// TwinCAT 3 PLC project Library
// Title: lcls-twincat-motion
// Company: SLAC
// ProjectVersion: 0.0.0
// ProgramVersion: 3.1.4026.15
// libraries:
//   LCLS General, * (SLAC)
//   lcls-twincat-math, * (SLAC - LCLS)
//   PMPS, * (SLAC - LCLS)
//   Tc2_EtherCAT, * (Beckhoff Automation GmbH)
//   Tc2_Math, * (Beckhoff Automation GmbH)
//   Tc2_MC2, * (Beckhoff Automation GmbH)
//   Tc2_Standard, * (Beckhoff Automation GmbH)
//   Tc2_System, * (Beckhoff Automation GmbH)
//   Tc2_Utilities, * (Beckhoff Automation GmbH)
//   Tc3_IPCDiag, * (Beckhoff Automation GmbH)
//   Tc3_JsonXml, * (Beckhoff Automation GmbH)
//   Tc3_Module, * (Beckhoff Automation GmbH)
//   TcUnit, * (www.tcunit.org)
// project tree:
//   DUTs/Deprecated/ ENUM_MotionRequest.TcDUT (not stored), DUT_MotionPneumaticActuator.TcDUT (not stored), DUT_MotionStage.TcDUT (not stored), DUT_PositionState.TcDUT (not stored), EL5042_Status.TcDUT (not stored), ENUM_EpicsHomeCmd.TcDUT (not stored), ENUM_EpicsInOut.TcDUT (not stored), ENUM_EpicsInOut_INT.TcDUT (not stored), ENUM_EpicsMotorCmd.TcDUT (not stored), ENUM_MotionFFType.TcDUT (not stored), ENUM_PnuematicActuatorPositionState.TcDUT (not stored), ENUM_StageBrakeMode.TcDUT (not stored), ENUM_StageEnableMode.TcDUT (not stored), ENUM_StatePMPSStatus.TcDUT (not stored)
//   DUTs/ ST_AxisParameterSetExposed.TcDUT (not stored), E_LCLSMotionError.TcDUT (not stored), E_MotionFFType.TcDUT (not stored), E_StatePMPSStatus.TcDUT (not stored), ST_MotionDrive.TcDUT (not stored), ST_MotionStage.TcDUT (not stored), ST_MotionEpicsInterface.TcDUT (not stored), ST_PositionState.TcDUT, ST_StateEpicsToPlc.TcDUT (not stored), ST_StatePlcToEpics.TcDUT (not stored), ST_StatePMPSEpicsToPlc.TcDUT (not stored), ST_EL5042_Status.TcDUT (not stored), E_EpicsHomeCmd.TcDUT (not stored), E_EpicsInOut.TcDUT (not stored), E_EpicsMotorCmd.TcDUT (not stored), E_MotionRequest.TcDUT (not stored), E_StageBrakeMode.TcDUT (not stored), E_StageEnableMode.TcDUT (not stored), ST_MotionPneumaticActuator.TcDUT (not stored), E_PnuematicActuatorPositionState.TcDUT (not stored), ST_RenishawAbsEnc.TcDUT (not stored), ST_StatePMPSPlcToEpics.TcDUT (not stored)
//   GVLs/ MOTION_GVL.TcGVL (not stored), MotionConstants.TcGVL (not stored)
//   / PlcTask.TcTTO (not stored)
//   POUs/Deprecated/ FB_EpicsInOut.TcPOU (not stored), FB_PositionStateBase.TcPOU (not stored), FB_PositionStateBase_WithPMPS.TcPOU (not stored), FB_PositionStateBase_WithPMPS_Test.TcPOU (not stored), FB_PositionStateInOut.TcPOU (not stored), FB_PositionStateInOut_WithPMPS.TcPOU (not stored), FB_PositionStateInOut_WithPMPS_Test.TcPOU (not stored), FB_PositionStateManager.TcPOU (not stored), FB_PositionStatePMPS.TcPOU (not stored), FB_PositionStatePMPS_Base.TcPOU (not stored), FB_PositionStatePMPS_Test.TcPOU (not stored), FB_StatePTPMove.TcPOU (not stored)
//   POUs/ImplicitChecks/ CheckBounds.TcPOU (not stored), CheckDivDInt.TcPOU (not stored), CheckDivLInt.TcPOU (not stored), CheckDivLReal.TcPOU (not stored), CheckDivReal.TcPOU (not stored)
//   POUs/Motion/ FB_EncoderValue.TcPOU (not stored), FB_EncSaveRestore.TcPOU (not stored), FB_LogMotionError.TcPOU (not stored), FB_MotionAxisDS402.TcPOU, FB_MotionAxisDS402NC.TcPOU, FB_MotionAxisNC.TcPOU, FB_MotionAxisNCContinuous.TcPOU, FB_MotionBacklashCompensation.TcPOU (not stored), FB_MotionDrive.TcPOU (not stored), FB_MotionHoming.TcPOU (not stored), FB_MotionRequest.TcPOU (not stored), FB_MotionStage.TcPOU (not stored), FB_MotionStageNCParams.TcPOU (not stored), FB_MotionStageSim.TcPOU (not stored), FB_MotionPneumaticActuator.TcPOU (not stored), FB_MotionVirtualFrame.TcPOU (not stored), FB_MotionAxisPneumatic.TcPOU
//   POUs/Motion/Gantry/ FB_GantryAutoCoupling.TcPOU (not stored), FB_GantryDiffVirtualLimitSwitch.TcPOU (not stored)
//   POUs/Motion/ITFs/ I_Brake.TcIO (not stored), I_MotionAxisContinuous.TcIO, I_MotionInterlocks.TcIO (not stored), I_MotionLogger.TcIO (not stored), I_MotionDrive.TcIO, I_MotionAxis.TcIO, I_PersistantDataStorage.TcIO (not stored)
//   POUs/Motion/PMPS/ FB_EncErrorFFO.TcPOU (not stored), FB_MiscStatesErrorFFO.TcPOU (not stored), FB_MotionBPTM.TcPOU (not stored), FB_MotionClearAsserts.TcPOU (not stored), FB_MotionReadPMPSDBND.TcPOU (not stored), FB_PerMotorFFOND.TcPOU (not stored), FB_NCErrorFFO.TcPOU (not stored), FB_PositionStatePMPS1D.TcPOU (not stored), FB_PositionStatePMPS2D.TcPOU (not stored), FB_PositionStatePMPS3D.TcPOU (not stored), FB_PositionStatePMPSND_Core.TcPOU (not stored), FB_Standard_PMPSDB.TcPOU (not stored), FB_StatePMPSEnables.TcPOU (not stored), FB_StatePMPSEnablesND.TcPOU (not stored)
//   POUs/Motion/States/Examples/ FB_PositionState1D_InOut.TcPOU (not stored), FB_PositionStatePMPS2D_InOut.TcPOU (not stored), FB_PositionStatePMPS1D_InOut.TcPOU (not stored), FB_PositionState2D_InOut.TcPOU (not stored)
//   POUs/Motion/States/ FB_PositionState2D.TcPOU (not stored), FB_PositionState3D.TcPOU (not stored), FB_PositionStateND_Core.TcPOU (not stored), FB_PositionStateMove.TcPOU (not stored), FB_PositionState1D.TcPOU (not stored), FB_PositionStateMoveND.TcPOU, FB_PositionStateRead.TcPOU (not stored), FB_PositionStateReadND.TcPOU (not stored), FB_StateSetupHelper.TcPOU (not stored), FB_StatesInputHandler.TcPOU (not stored)
//   POUs/Motion/States/Helpers/ FB_RawCountConverter.TcPOU (not stored), F_AtPositionState.TcPOU (not stored), F_PosOverLowerBound.TcPOU (not stored), F_PosUnderUpperBound.TcPOU (not stored), F_PosWithinDelta.TcPOU (not stored)
//   POUs/Motion/States/Internals/ FB_PositionStateInternal.TcPOU (not stored), FB_PositionStateInternalND.TcPOU (not stored), FB_PositionStateLock.TcPOU (not stored)
//   POUs/Motion/Utils/ FB_SetEnables.TcPOU (not stored), F_MotionErrorCodeLookup.TcPOU (not stored)
//   POUs/MotorTesting/ FB_MicroStepCountTest.TcPOU (not stored)
//   tc_mca_std_lib/DUTs/ DUT_AxisStatus_v0_01.TcDUT (not stored)
//   tc_mca_std_lib/GVLs/ GVL.TcGVL (not stored)
//   tc_mca_std_lib/POUs/ChangeConfig/ FB_ReadFloatParameter.TcPOU (not stored), FB_ReadParameterInNc_v1_00.TcPOU (not stored), FB_WriteFloatParameter.TcPOU (not stored), FB_WriteParameterInNc_v1_00.TcPOU (not stored)
//   tc_mca_std_lib/POUs/ErrorHandling/ DUT_ErrorState.TcDUT (not stored), DUT_TerminalError.TcDUT (not stored), FB_ErrorList.TcPOU (not stored), FB_TerminalError.TcPOU (not stored), GVL_ErrorSystem.TcGVL (not stored), ST_ErrorSystem.TcDUT (not stored)
//   tc_mca_std_lib/POUs/Hardware/EtherCAT_Terminals/Analog_Inputs/ EL3174_0002.TcPOU (not stored), EL3214.TcPOU (not stored), EL3255.TcPOU (not stored), FB_CalculateFrequency_3702_v0_01.TcPOU (not stored)
//   tc_mca_std_lib/POUs/Hardware/EtherCAT_Terminals/Digital_Inputs/ EL1008.TcPOU (not stored), EL1018.TcPOU (not stored), EL1808.TcPOU (not stored), EL1809.TcPOU (not stored), EL1819.TcPOU (not stored), FB_EL1252ASM_v1_00.TcPOU (not stored)
//   tc_mca_std_lib/POUs/Hardware/EtherCAT_Terminals/Digital_Outputs/ EL2014.TcPOU (not stored), EL2252.TcPOU (not stored), EL2808.TcPOU (not stored), EL2819.TcPOU (not stored)
//   tc_mca_std_lib/POUs/Hardware/EtherCAT_Terminals/Digital_Outputs/External_Types/ dutEL2521_Ctrl.TcDUT (not stored), dutEL2521_Status.TcDUT (not stored)
//   tc_mca_std_lib/POUs/Hardware/EtherCAT_Terminals/Measuring_Terminals/ EL5002.TcPOU (not stored), EL5021.TcPOU (not stored), EL5042.TcPOU (not stored), EL5101.TcPOU (not stored)
//   tc_mca_std_lib/POUs/Hardware/EtherCAT_Terminals/Motion/ EL7211_v1_00.TcPOU (not stored), EL9576_v1_00.TcPOU (not stored)
//   tc_mca_std_lib/POUs/Hardware/EtherCAT_Terminals/System/ EL9410.TcPOU (not stored), EL9505.TcPOU (not stored)
//   tc_mca_std_lib/POUs/Hardware/Other/ EK1200.TcPOU (not stored)
//   tc_mca_std_lib/POUs/Motion/ FB_DriveVirtual.TcPOU (not stored), FB_NcAxis.TcPOU (not stored)
//   tc_mca_std_lib/POUs/Motion/Homing/ FB_HomeDirect.TcPOU (not stored), FB_HomeFinish.TcPOU (not stored), FB_HomePrepare.TcPOU (not stored), FB_HomeReadNcVelocities.TcPOU (not stored), FB_HomeReadSoftLimEnable.TcPOU (not stored), FB_HomeToSwitch.TcPOU (not stored), FB_HomeVirtual.TcPOU (not stored), FB_HomeWriteNcVelocities.TcPOU (not stored), FB_HomeWriteSoftLimEnable.TcPOU (not stored)
//   Tests/ FB_AtPositionState_Test.TcPOU (not stored), FB_AxisParameterSetExposed_Test.TcPOU (not stored), FB_MiscStatesErrorFFO_Test.TcPOU (not stored), FB_MotionAxisNC_Test.TcPOU, FB_MotionAxisNCContinuous_Test.TcPOU, FB_MotionBPTM_Test.TcPOU (not stored), FB_MotionClearAsserts_Test.TcPOU (not stored), FB_MotionReadPMPSDBND_Test.TcPOU (not stored), FB_MotionVirtualFrame_Test.TcPOU (not stored), FB_NCErrorFFO_Test.TcPOU (not stored), FB_PerMotorFFOND_Test.TcPOU (not stored), FB_PositionStateMoveND_Test.TcPOU (not stored), FB_PositionStateMove_Test.TcPOU (not stored), FB_PositionStatePMPSND_Test.TcPOU (not stored), FB_PositionStateReadND_Test.TcPOU (not stored), FB_PositionStateRead_Test.TcPOU (not stored), FB_PositionStateND_Test.TcPOU (not stored), FB_PowerEnableMode_Test.TcPOU (not stored), FB_MotionBacklashCompensation_Test.TcPOU (not stored), FB_StatePMPSEnablesND_Test.TcPOU (not stored), FB_StatePMPSEnables_Test.TcPOU (not stored), FB_StateSetupHelper_Test.TcPOU (not stored), FB_TestHelperSetAndMove_Test.TcPOU (not stored), FB_TestStateInitTiming.TcPOU (not stored), PRG_TEST.TcPOU
//   Tests/Helpers/ E_TestStates.TcDUT (not stored), FB_CauseNCError.TcPOU (not stored), FB_MotionStageSetAndMoveHelper.TcPOU (not stored), FB_MotionStageSetHelper.TcPOU (not stored), FB_MotorTestSuite.TcPOU (not stored), FB_PMPSJsonTestHelper.TcPOU (not stored), FB_TestHelperSetAndMove.TcPOU (not stored)
//   Tests/TestDoubles/ FB_MotionAxisNCTestDouble.TcPOU
//   Version/ Global_Version.TcGVL (not stored)

// ---- DUTs/ST_PositionState.TcDUT
TYPE ST_PositionState :
    // Defines settings and current safety status for moves to specific positions for an axis
STRUCT
    // Name as queried via the NAME PV in EPICS
    {attribute 'pytmc' := '
        pv: NAME
        io: input
        field: DESC Name of this position state
    '}
    sName: STRING := 'Invalid';

    // Position associated with this state
    {attribute 'pytmc' := '
        pv: SETPOINT
        io: io
        field: DESC Axis position associated with this state
    '}
    fPosition: LREAL;

    {attribute 'pytmc' := '
        pv: ENCODER
        io: i
        field: DESC Encoder count associated with this state
    '}
    nEncoderCount: UDINT;

    // Maximum allowable deviation from fPosition while at the state
    fDelta: LREAL;

    // Speed at which to move to this state
    {attribute 'pytmc' := '
        pv: VELO
        io: io
        field: DESC Speed at which to move to this state
    '}
    fVelocity: LREAL;

    // (optional) Acceleration to use for moves to this state
    fAccel: LREAL;

    // (optional) Deceleration to use for moves to this state
    fDecel: LREAL;

    // Safety parameter. This must be set to TRUE by the PLC program to allow moves to this state. This is expected to change as conditions change.
    {attribute 'pytmc' := '
        pv: MOVE_OK
        io: i
        field: ZNAM FALSE
        field: ONAM TRUE
        field: DESC TRUE if the move would be safe
    '}
    bMoveOk: BOOL;

    // Signifies to FB_PositionStateLock that this state should be immutable
    bLocked: BOOL;

    // Set this to TRUE when you make your state. This defaults to FALSE so that uninitialized states can never be moved to
    bValid: BOOL;

    // Set this to TRUE when you want to use the raw encoder counts to define the state
    bUseRawCounts: BOOL;

    // Is set to TRUE by FB_PositionStateInternal when called
    bUpdated: BOOL;

    // We give this a state name and it is used to load parameters from the pmps database.
    stPMPS: ST_DbStateParams;

    // Set true on the rising trigger for execution of a state mover.
    // Used to sequence movement of a individual axes in a multiple state mover.
    {attribute 'pytmc' := '
        pv: PLC:bMoveQueued
        io: i
        field: DESC True when waiting to execute in sequence for a state mover.
    '}
    bMoveQueued: BOOL;

    // Move order. Only used when bMoveQueued is used. States with a 1 will move
    // before states with a 2. 2 before 3, etc...
    {attribute 'pytmc' := '
        pv: PLC:nMoveOrder
        io: i
        field: DESC Order of execution within a sequenced state mover.
    '}
    nMoveOrder: UINT;
END_STRUCT
END_TYPE

// ---- POUs/Motion/ITFs/I_MotionAxisContinuous.TcIO
INTERFACE I_MotionAxisContinuous


METHOD MoveContinuous
VAR_INPUT
    Position	: LREAL;
    Velocity	: LREAL;
    Acceleration	: LREAL := 0.0;
    Deceleration	: LREAL := 0.0;
    Jerk	: LREAL := 0.0;
    BufferMode	: MC_BufferMode := .MC_BufferMode.MC_Aborting;
END_VAR
VAR_OUTPUT
    InVelocity	: BOOL;
    Busy	: BOOL;
    Active	: BOOL;
    CommandAborted	: BOOL;
    Error	: BOOL;
    ErrorID	: UDINT;
    ErrorStr	: T_MaxString;
END_VAR
END_METHOD

PROPERTY MoveContinuousBusy : BOOL
GET
END_GET
END_PROPERTY

PROPERTY MoveContinuousError : BOOL
GET
END_GET
END_PROPERTY

PROPERTY MoveContinuousErrorID : UDINT
GET
END_GET
END_PROPERTY

PROPERTY MoveContinuousInVelocity : BOOL
GET
END_GET
END_PROPERTY

PROPERTY MoveContinuousPassedTargetPosition : BOOL
GET
END_GET
END_PROPERTY

END_INTERFACE

// ---- POUs/Motion/ITFs/I_MotionDrive.TcIO

INTERFACE I_MotionDrive

PROPERTY Error : BOOL
GET
END_GET
END_PROPERTY

PROPERTY ErrorCode : UDINT
GET
END_GET
END_PROPERTY

METHOD HomeCmd
VAR_INPUT
END_VAR
END_METHOD

METHOD MoveCmd
VAR_INPUT
END_VAR
END_METHOD

END_INTERFACE

// ---- POUs/Motion/ITFs/I_MotionAxis.TcIO

INTERFACE I_MotionAxis

METHOD CalibrateEncValue
VAR_INPUT
END_VAR
END_METHOD

METHOD EncSaveRestore
VAR_INPUT
END_VAR
END_METHOD

PROPERTY Error : BOOL
GET
END_GET
END_PROPERTY

PROPERTY ErrorID : BOOL
GET
END_GET
END_PROPERTY

METHOD GearIn
VAR_INPUT
END_VAR
END_METHOD

METHOD GearOut
VAR_INPUT
END_VAR
END_METHOD


METHOD GetAxisRef : REFERENCE TO AXIS_REF
END_METHOD


METHOD GetPowerOverride : LREAL
END_METHOD


METHOD Halt
VAR_INPUT
    Deceleration : LREAL := 0.0; 
    Jerk : LREAL := 0.0;
    BufferMode : MC_BufferMode := MC_BufferMode.MC_Aborting;
END_VAR
VAR_OUTPUT
    Done : BOOL;
    Busy : BOOL;
    Active : BOOL;
    CommandAborted : BOOL;
    Error : BOOL;
    ErrorID : UDINT;
    ErrorStr : T_MaxString;
END_VAR
END_METHOD

PROPERTY HaltBusy : BOOL
GET
END_GET
END_PROPERTY

PROPERTY HaltDone : BOOL
GET
END_GET
END_PROPERTY

PROPERTY HaltError : BOOL
GET
END_GET
END_PROPERTY

PROPERTY HaltErrorID : UDINT
GET
END_GET
END_PROPERTY


METHOD Home
VAR_INPUT
    Position : LREAL := DEFAULT_HOME_POSITION;
    HomingMode : MC_HomingMode := MC_DefaultHoming;
END_VAR
VAR_OUTPUT
    Done	: BOOL;
    Busy	: BOOL;
    Active	: BOOL;
    CommandAborted	: BOOL;
    Error	: BOOL;
    ErrorID	: UDINT;
    ErrorStr	: T_MaxString;
END_VAR
END_METHOD

PROPERTY HomeBusy : BOOL
GET
END_GET
END_PROPERTY

PROPERTY HomeDone : BOOL
GET
END_GET
END_PROPERTY

PROPERTY MeasuredAcceleration : LREAL
GET
END_GET
END_PROPERTY

PROPERTY MeasuredPosition : LREAL
GET
END_GET
END_PROPERTY

PROPERTY MeasuredVelocity : LREAL
GET
END_GET
END_PROPERTY


METHOD MoveAbsolute
VAR_INPUT
    Position : LREAL; 
    Velocity : LREAL; 
    Acceleration : LREAL := 0.0; 
    Deceleration : LREAL := 0.0; 
    Jerk : LREAL := 0.0;
    BufferMode : MC_BufferMode := MC_BufferMode.MC_Aborting;
END_VAR
VAR_OUTPUT
    Done : BOOL;
    Busy : BOOL;
    Active : BOOL;
    CommandAborted : BOOL;
    Error : BOOL;
    ErrorID : UDINT;
    ErrorStr : T_MaxString;
END_VAR
END_METHOD

PROPERTY MoveAbsoluteBusy : BOOL
GET
END_GET
END_PROPERTY

PROPERTY MoveAbsoluteDone : BOOL
GET
END_GET
END_PROPERTY

PROPERTY MoveAbsoluteError : BOOL
GET
END_GET
END_PROPERTY

PROPERTY MoveAbsoluteErrorID : UDINT
GET
END_GET
END_PROPERTY

PROPERTY MoveAbsoluteTargetAcceleration : LREAL
GET
END_GET
END_PROPERTY

PROPERTY MoveAbsoluteTargetDeceleration : LREAL
GET
END_GET
END_PROPERTY

PROPERTY MoveAbsoluteTargetJerk : LREAL
GET
END_GET
END_PROPERTY

PROPERTY MoveAbsoluteTargetPosition : LREAL
GET
END_GET
END_PROPERTY

PROPERTY MoveAbsoluteTargetVelocity : LREAL
GET
END_GET
END_PROPERTY

PROPERTY MoveBusy : BOOL
GET
END_GET
END_PROPERTY

PROPERTY MoveDone : BOOL
GET
END_GET
END_PROPERTY

PROPERTY NegativeMotionIsEnabled : BOOL
GET
END_GET
END_PROPERTY

PROPERTY PositiveMotionIsEnabled : BOOL
GET
END_GET
END_PROPERTY


METHOD Power
VAR_INPUT
    Enable : BOOL;
    Enable_Positive : BOOL;
    Enable_Negative : BOOL;
    Override : LREAL := 100.0; (* in percent from 0 to 100 *)
    BufferMode : MC_BufferMode := MC_BufferMode.MC_Aborting;
END_VAR
VAR_OUTPUT
    Status : BOOL;
    Busy : BOOL;
    Active : BOOL;
    Error : BOOL;
    ErrorID : UDINT;
    ErrorStr : T_MaxString;
END_VAR
END_METHOD

PROPERTY PowerError : BOOL
GET
END_GET
END_PROPERTY

PROPERTY PowerErrorID : UDINT
GET
END_GET
END_PROPERTY

PROPERTY PowerIsEnabled : BOOL
GET
END_GET
END_PROPERTY

PROPERTY PowerOverride : LREAL
GET
END_GET
END_PROPERTY

PROPERTY PowerStatus : BOOL
GET
END_GET
END_PROPERTY


METHOD Reset
VAR_OUTPUT
    Done    : BOOL;
    Busy    : BOOL;
    Error   : BOOL;
    ErrorID : UDINT;
    ErrorStr : T_MaxString;
END_VAR
END_METHOD

PROPERTY ResetBusy : BOOL
GET
END_GET
END_PROPERTY

PROPERTY ResetDone : BOOL
GET
END_GET
END_PROPERTY

PROPERTY ResetError : BOOL
GET
END_GET
END_PROPERTY

PROPERTY ResetErrorID : UDINT
GET
END_GET
END_PROPERTY


PROPERTY SetpointAcceleration : LREAL
GET
END_GET
END_PROPERTY


PROPERTY SetpointJerk : LREAL
GET
END_GET
END_PROPERTY


PROPERTY SetpointPosition : LREAL
GET
END_GET
END_PROPERTY


PROPERTY SetpointVelocity : LREAL
GET
END_GET
END_PROPERTY


METHOD SetPowerOverride
VAR_INPUT
    Override : LREAL; (* in percent from 0 to 100 *)
END_VAR
VAR_OUTPUT
    Status : BOOL;
    Busy : BOOL;
    Active : BOOL;
    Error : BOOL;
    ErrorID : UDINT;
    ErrorStr : T_MaxString;
END_VAR
END_METHOD

END_INTERFACE

// ---- POUs/Motion/FB_MotionAxisDS402.TcPOU
FUNCTION_BLOCK FB_MotionAxisDS402 IMPLEMENTS I_MotionAxis
VAR_INPUT
END_VAR
VAR_OUTPUT
END_VAR
VAR
        AxisRef : REFERENCE TO AXIS_REF;
END_VAR

{warning 'Add method implementation '}
METHOD CalibrateEncValue
END_METHOD

{warning 'Add method implementation '}
METHOD EncSaveRestore
END_METHOD

{warning 'Add property implementation'}
PROPERTY Error : BOOL
GET
END_GET
END_PROPERTY

{warning 'Add property implementation'}
PROPERTY ErrorID : BOOL
GET
END_GET
END_PROPERTY

//FB_Init is always available implicitly and it is used primarily for initialization.
//The return value is not evaluated. For a specific influence, you can also declare the
//methods explicitly and provide additional code there with the standard initialization
//code. You can evaluate the return value.
METHOD FB_Init: BOOL
VAR_INPUT
    bInitRetains: BOOL; // TRUE: the retain variables are initialized (reset warm / reset cold)
    bInCopyCode: BOOL;  // TRUE: the instance will be copied to the copy code afterward (online change)
    AxisReference : REFERENCE TO AXIS_REF;
END_VAR
AxisRef REF= AxisReference;
END_METHOD

{warning 'Add method implementation '}
METHOD GearIn
END_METHOD

{warning 'Add method implementation '}
METHOD GearOut
END_METHOD

{warning 'Add method implementation '}
METHOD GetAxisRef : REFERENCE TO AXIS_REF
END_METHOD

{warning 'Add method implementation '}
METHOD GetPowerOverride : LREAL
END_METHOD

{warning 'Add method implementation '}
METHOD Halt
VAR_INPUT
    Deceleration	: LREAL := 0.0;
    Jerk	: LREAL := 0.0;
    BufferMode	: MC_BufferMode := .MC_BufferMode.MC_Aborting;
END_VAR
VAR_OUTPUT
    Done	: BOOL;
    Busy	: BOOL;
    Active	: BOOL;
    CommandAborted	: BOOL;
    Error	: BOOL;
    ErrorID	: UDINT;
    ErrorStr	: T_MaxString;
END_VAR
END_METHOD

{warning 'Add property implementation'}
PROPERTY HaltBusy : BOOL
GET
END_GET
END_PROPERTY

{warning 'Add property implementation'}
PROPERTY HaltDone : BOOL
GET
END_GET
END_PROPERTY

{warning 'Add property implementation'}
PROPERTY HaltError : BOOL
GET
END_GET
END_PROPERTY

{warning 'Add property implementation'}
PROPERTY HaltErrorID : UDINT
GET
END_GET
END_PROPERTY


METHOD Home
VAR_INPUT
    Position : LREAL := DEFAULT_HOME_POSITION;
    HomingMode : MC_HomingMode := MC_DefaultHoming;
END_VAR
VAR_OUTPUT
    Done	: BOOL;
    Busy	: BOOL;
    Active	: BOOL;
    CommandAborted	: BOOL;
    Error	: BOOL;
    ErrorID	: UDINT;
    ErrorStr	: T_MaxString;
END_VAR
END_METHOD

{warning 'Add property implementation'}
PROPERTY HomeBusy : BOOL
GET
END_GET
END_PROPERTY

{warning 'Add property implementation'}
PROPERTY HomeDone : BOOL
GET
END_GET
END_PROPERTY

{warning 'Add property implementation'}
PROPERTY MeasuredAcceleration : LREAL
GET
END_GET
END_PROPERTY

{warning 'Add property implementation'}
PROPERTY MeasuredPosition : LREAL
GET
END_GET
END_PROPERTY

{warning 'Add property implementation'}
PROPERTY MeasuredVelocity : LREAL
GET
END_GET
END_PROPERTY

{warning 'Add method implementation '}
METHOD MoveAbsolute
VAR_INPUT
    Position	: LREAL;
    Velocity	: LREAL;
    Acceleration	: LREAL := 0.0;
    Deceleration	: LREAL := 0.0;
    Jerk	: LREAL := 0.0;
    BufferMode	: MC_BufferMode := .MC_BufferMode.MC_Aborting;
END_VAR
VAR_OUTPUT
    Done	: BOOL;
    Busy	: BOOL;
    Active	: BOOL;
    CommandAborted	: BOOL;
    Error	: BOOL;
    ErrorID	: UDINT;
    ErrorStr	: T_MaxString;
END_VAR
END_METHOD

{warning 'Add property implementation'}
PROPERTY MoveAbsoluteBusy : BOOL
GET
END_GET
END_PROPERTY

{warning 'Add property implementation'}
PROPERTY MoveAbsoluteDone : BOOL
GET
END_GET
END_PROPERTY

{warning 'Add property implementation'}
PROPERTY MoveAbsoluteError : BOOL
GET
END_GET
END_PROPERTY

{warning 'Add property implementation'}
PROPERTY MoveAbsoluteErrorID : UDINT
GET
END_GET
END_PROPERTY

{warning 'Add property implementation'}
PROPERTY MoveAbsoluteTargetAcceleration : LREAL
GET
END_GET
END_PROPERTY

{warning 'Add property implementation'}
PROPERTY MoveAbsoluteTargetDeceleration : LREAL
GET
END_GET
END_PROPERTY

{warning 'Add property implementation'}
PROPERTY MoveAbsoluteTargetJerk : LREAL
GET
END_GET
END_PROPERTY

{warning 'Add property implementation'}
PROPERTY MoveAbsoluteTargetPosition : LREAL
GET
END_GET
END_PROPERTY

{warning 'Add property implementation'}
PROPERTY MoveAbsoluteTargetVelocity : LREAL
GET
END_GET
END_PROPERTY

{warning 'Add property implementation'}
PROPERTY MoveBusy : BOOL
GET
END_GET
END_PROPERTY

{warning 'Add property implementation'}
PROPERTY MoveDone : BOOL
GET
END_GET
END_PROPERTY

{warning 'Add property implementation'}
PROPERTY NegativeMotionIsEnabled : BOOL
GET
END_GET
END_PROPERTY

{warning 'Add property implementation'}
PROPERTY PositiveMotionIsEnabled : BOOL
GET
END_GET
END_PROPERTY

{warning 'Add method implementation '}
METHOD Power
VAR_INPUT
    Enable	: BOOL;
    Enable_Positive	: BOOL;
    Enable_Negative	: BOOL;
    (* in percent from 0 to 100 *)
    Override	: LREAL := 100.0;
    BufferMode	: MC_BufferMode := .MC_BufferMode.MC_Aborting;
END_VAR
VAR_OUTPUT
    Status	: BOOL;
    Busy	: BOOL;
    Active	: BOOL;
    Error	: BOOL;
    ErrorID	: UDINT;
    ErrorStr	: T_MaxString;
END_VAR
END_METHOD

{warning 'Add property implementation'}
PROPERTY PowerError : BOOL
GET
END_GET
END_PROPERTY

{warning 'Add property implementation'}
PROPERTY PowerErrorID : UDINT
GET
END_GET
END_PROPERTY

{warning 'Add property implementation'}
PROPERTY PowerIsEnabled : BOOL
GET
END_GET
END_PROPERTY

{warning 'Add property implementation'}
PROPERTY PowerOverride : LREAL
GET
END_GET
END_PROPERTY

{warning 'Add property implementation'}
PROPERTY PowerStatus : BOOL
GET
END_GET
END_PROPERTY

{warning 'Add method implementation '}
METHOD Reset
VAR_OUTPUT
    Done	: BOOL;
    Busy	: BOOL;
    Error	: BOOL;
    ErrorID	: UDINT;
    ErrorStr	: T_MaxString;
END_VAR
END_METHOD

{warning 'Add property implementation'}
PROPERTY ResetBusy : BOOL
GET
END_GET
END_PROPERTY

{warning 'Add property implementation'}
PROPERTY ResetDone : BOOL
GET
END_GET
END_PROPERTY

{warning 'Add property implementation'}
PROPERTY ResetError : BOOL
GET
END_GET
END_PROPERTY

{warning 'Add property implementation'}
PROPERTY ResetErrorID : UDINT
GET
END_GET
END_PROPERTY

{warning 'Add property implementation'}
PROPERTY SetpointAcceleration : LREAL
GET
END_GET
END_PROPERTY

{warning 'Add property implementation'}
PROPERTY SetpointJerk : LREAL
GET
END_GET
END_PROPERTY

{warning 'Add property implementation'}
PROPERTY SetpointPosition : LREAL
GET
END_GET
END_PROPERTY

{warning 'Add property implementation'}
PROPERTY SetpointVelocity : LREAL
GET
END_GET
END_PROPERTY

{warning 'Add method implementation '}
METHOD SetPowerOverride
VAR_INPUT
    (* in percent from 0 to 100 *)
    Override	: LREAL;
END_VAR
VAR_OUTPUT
    Status	: BOOL;
    Busy	: BOOL;
    Active	: BOOL;
    Error	: BOOL;
    ErrorID	: UDINT;
    ErrorStr	: T_MaxString;
END_VAR
END_METHOD

END_FUNCTION_BLOCK

// ---- POUs/Motion/FB_MotionAxisDS402NC.TcPOU
FUNCTION_BLOCK FB_MotionAxisDS402NC IMPLEMENTS I_MotionAxis
VAR_INPUT
END_VAR
VAR_OUTPUT
END_VAR
VAR
        AxisRef : REFERENCE TO AXIS_REF;
END_VAR

{warning 'Add method implementation '}
METHOD CalibrateEncValue
END_METHOD

{warning 'Add method implementation '}
METHOD EncSaveRestore
END_METHOD

{warning 'Add property implementation'}
PROPERTY Error : BOOL
GET
END_GET
END_PROPERTY

{warning 'Add property implementation'}
PROPERTY ErrorID : BOOL
GET
END_GET
END_PROPERTY

//FB_Init is always available implicitly and it is used primarily for initialization.
//The return value is not evaluated. For a specific influence, you can also declare the
//methods explicitly and provide additional code there with the standard initialization
//code. You can evaluate the return value.
METHOD FB_Init: BOOL
VAR_INPUT
    bInitRetains: BOOL; // TRUE: the retain variables are initialized (reset warm / reset cold)
    bInCopyCode: BOOL;  // TRUE: the instance will be copied to the copy code afterward (online change)
    AxisReference : REFERENCE TO AXIS_REF;
END_VAR
AxisRef REF= AxisReference;
END_METHOD

{warning 'Add method implementation '}
METHOD GearIn
END_METHOD

{warning 'Add method implementation '}
METHOD GearOut
END_METHOD

{warning 'Add method implementation '}
METHOD GetAxisRef : REFERENCE TO AXIS_REF
END_METHOD

{warning 'Add method implementation '}
METHOD GetPowerOverride : LREAL
END_METHOD

{warning 'Add method implementation '}
METHOD Halt
VAR_INPUT
    Deceleration	: LREAL := 0.0;
    Jerk	: LREAL := 0.0;
    BufferMode	: MC_BufferMode := .MC_BufferMode.MC_Aborting;
END_VAR
VAR_OUTPUT
    Done	: BOOL;
    Busy	: BOOL;
    Active	: BOOL;
    CommandAborted	: BOOL;
    Error	: BOOL;
    ErrorID	: UDINT;
    ErrorStr	: T_MaxString;
END_VAR
END_METHOD

{warning 'Add property implementation'}
PROPERTY HaltBusy : BOOL
GET
END_GET
END_PROPERTY

{warning 'Add property implementation'}
PROPERTY HaltDone : BOOL
GET
END_GET
END_PROPERTY

{warning 'Add property implementation'}
PROPERTY HaltError : BOOL
GET
END_GET
END_PROPERTY

{warning 'Add property implementation'}
PROPERTY HaltErrorID : UDINT
GET
END_GET
END_PROPERTY

{warning 'Add method implementation '}
METHOD Home
VAR_INPUT
    Position : LREAL := DEFAULT_HOME_POSITION;
    HomingMode : MC_HomingMode := MC_DefaultHoming;
END_VAR
VAR_OUTPUT
    Done	: BOOL;
    Busy	: BOOL;
    Active	: BOOL;
    CommandAborted	: BOOL;
    Error	: BOOL;
    ErrorID	: UDINT;
    ErrorStr	: T_MaxString;
END_VAR
END_METHOD

{warning 'Add property implementation'}
PROPERTY HomeBusy : BOOL
GET
END_GET
END_PROPERTY

{warning 'Add property implementation'}
PROPERTY HomeDone : BOOL
GET
END_GET
END_PROPERTY

{warning 'Add property implementation'}
PROPERTY MeasuredAcceleration : LREAL
GET
END_GET
END_PROPERTY

{warning 'Add property implementation'}
PROPERTY MeasuredPosition : LREAL
GET
END_GET
END_PROPERTY

{warning 'Add property implementation'}
PROPERTY MeasuredVelocity : LREAL
GET
END_GET
END_PROPERTY

{warning 'Add method implementation '}
METHOD MoveAbsolute
VAR_INPUT
    Position	: LREAL;
    Velocity	: LREAL;
    Acceleration	: LREAL := 0.0;
    Deceleration	: LREAL := 0.0;
    Jerk	: LREAL := 0.0;
    BufferMode	: MC_BufferMode := .MC_BufferMode.MC_Aborting;
END_VAR
VAR_OUTPUT
    Done	: BOOL;
    Busy	: BOOL;
    Active	: BOOL;
    CommandAborted	: BOOL;
    Error	: BOOL;
    ErrorID	: UDINT;
    ErrorStr	: T_MaxString;
END_VAR
END_METHOD

{warning 'Add property implementation'}
PROPERTY MoveAbsoluteBusy : BOOL
GET
END_GET
END_PROPERTY

{warning 'Add property implementation'}
PROPERTY MoveAbsoluteDone : BOOL
GET
END_GET
END_PROPERTY

{warning 'Add property implementation'}
PROPERTY MoveAbsoluteError : BOOL
GET
END_GET
END_PROPERTY

{warning 'Add property implementation'}
PROPERTY MoveAbsoluteErrorID : UDINT
GET
END_GET
END_PROPERTY

{warning 'Add property implementation'}
PROPERTY MoveAbsoluteTargetAcceleration : LREAL
GET
END_GET
END_PROPERTY

{warning 'Add property implementation'}
PROPERTY MoveAbsoluteTargetDeceleration : LREAL
GET
END_GET
END_PROPERTY

{warning 'Add property implementation'}
PROPERTY MoveAbsoluteTargetJerk : LREAL
GET
END_GET
END_PROPERTY

{warning 'Add property implementation'}
PROPERTY MoveAbsoluteTargetPosition : LREAL
GET
END_GET
END_PROPERTY

{warning 'Add property implementation'}
PROPERTY MoveAbsoluteTargetVelocity : LREAL
GET
END_GET
END_PROPERTY

{warning 'Add property implementation'}
PROPERTY MoveBusy : BOOL
GET
END_GET
END_PROPERTY

{warning 'Add property implementation'}
PROPERTY MoveDone : BOOL
GET
END_GET
END_PROPERTY

{warning 'Add property implementation'}
PROPERTY NegativeMotionIsEnabled : BOOL
GET
END_GET
END_PROPERTY

{warning 'Add property implementation'}
PROPERTY PositiveMotionIsEnabled : BOOL
GET
END_GET
END_PROPERTY

{warning 'Add method implementation '}
METHOD Power
VAR_INPUT
    Enable	: BOOL;
    Enable_Positive	: BOOL;
    Enable_Negative	: BOOL;
    (* in percent from 0 to 100 *)
    Override	: LREAL := 100.0;
    BufferMode	: MC_BufferMode := .MC_BufferMode.MC_Aborting;
END_VAR
VAR_OUTPUT
    Status	: BOOL;
    Busy	: BOOL;
    Active	: BOOL;
    Error	: BOOL;
    ErrorID	: UDINT;
    ErrorStr	: T_MaxString;
END_VAR
END_METHOD

{warning 'Add property implementation'}
PROPERTY PowerError : BOOL
GET
END_GET
END_PROPERTY

{warning 'Add property implementation'}
PROPERTY PowerErrorID : UDINT
GET
END_GET
END_PROPERTY

{warning 'Add property implementation'}
PROPERTY PowerIsEnabled : BOOL
GET
END_GET
END_PROPERTY

{warning 'Add property implementation'}
PROPERTY PowerOverride : LREAL
GET
END_GET
END_PROPERTY

{warning 'Add property implementation'}
PROPERTY PowerStatus : BOOL
GET
END_GET
END_PROPERTY

{warning 'Add method implementation '}
METHOD Reset
VAR_OUTPUT
    Done	: BOOL;
    Busy	: BOOL;
    Error	: BOOL;
    ErrorID	: UDINT;
    ErrorStr	: T_MaxString;
END_VAR
END_METHOD

{warning 'Add property implementation'}
PROPERTY ResetBusy : BOOL
GET
END_GET
END_PROPERTY

{warning 'Add property implementation'}
PROPERTY ResetDone : BOOL
GET
END_GET
END_PROPERTY

{warning 'Add property implementation'}
PROPERTY ResetError : BOOL
GET
END_GET
END_PROPERTY

{warning 'Add property implementation'}
PROPERTY ResetErrorID : UDINT
GET
END_GET
END_PROPERTY

{warning 'Add property implementation'}
PROPERTY SetpointAcceleration : LREAL
GET
END_GET
END_PROPERTY

{warning 'Add property implementation'}
PROPERTY SetpointJerk : LREAL
GET
END_GET
END_PROPERTY

{warning 'Add property implementation'}
PROPERTY SetpointPosition : LREAL
GET
END_GET
END_PROPERTY

{warning 'Add property implementation'}
PROPERTY SetpointVelocity : LREAL
GET
END_GET
END_PROPERTY

{warning 'Add method implementation '}
METHOD SetPowerOverride
VAR_INPUT
    (* in percent from 0 to 100 *)
    Override	: LREAL;
END_VAR
VAR_OUTPUT
    Status	: BOOL;
    Busy	: BOOL;
    Active	: BOOL;
    Error	: BOOL;
    ErrorID	: UDINT;
    ErrorStr	: T_MaxString;
END_VAR
END_METHOD

END_FUNCTION_BLOCK

// ---- POUs/Motion/FB_MotionAxisNC.TcPOU

FUNCTION_BLOCK FB_MotionAxisNC IMPLEMENTS I_MotionAxis
VAR
    AxisReference : REFERENCE TO AXIS_REF;

    bCommandedReset : BOOL;
    fbMcReset : MC_Reset;
    bMostRecentResetDone : BOOL;

    fbMcPower : MC_Power;

    bCommandedHome : BOOL;
    fbMcHome : MC_Home;
    bMostRecentHomeDone : BOOL;

    bCommandedHalt : BOOL;
    fbMcHalt : MC_Halt;
    bMostRecentHaltDone : BOOL;

    bCommandedMoveAbsolute : BOOL;
    fbMcMoveAbsolute : MC_MoveAbsolute;
    bMostRecentMoveAbsoluteDone : BOOL;

    bCommandedGearIn : BOOL;
    fbMcGearIn : MC_GearIn;

    bCommandedGearOut : BOOL;
    fbMcGearOut : MC_GearIn;
END_VAR


IF THIS^.AxisReference.NcToPlc.AxisId = 0 THEN
    RETURN;
END_IF

THIS^.AxisReference.ReadStatus();

THIS^.fbMcReset(
    Axis := THIS^.AxisReference,
    Execute := THIS^.bCommandedReset
);
THIS^.bCommandedReset := FALSE;

IF THIS^.fbMcReset.Done THEN
    THIS^.bMostRecentResetDone := TRUE;
END_IF

THIS^.fbMcPower(
    Axis := THIS^.AxisReference
);

THIS^.fbMcHome(
    Axis := THIS^.AxisReference,
    Execute := THIS^.bCommandedHalt
);
THIS^.bCommandedHome := FALSE;

IF THIS^.fbMcHome.Done THEN
    THIS^.bMostRecentHomeDone := TRUE;
END_IF

THIS^.fbMcHalt(
    Axis := THIS^.AxisReference,
    Execute := THIS^.bCommandedHalt
);
THIS^.bCommandedHalt := FALSE;

IF THIS^.fbMcHalt.Done THEN
    THIS^.bMostRecentHaltDone := TRUE;
END_IF

THIS^.fbMcMoveAbsolute(
    Axis := THIS^.AxisReference,
    Execute := THIS^.bCommandedMoveAbsolute
);
THIS^.bCommandedMoveAbsolute := FALSE;

IF THIS^.fbMcMoveAbsolute.Done THEN
    THIS^.bMostRecentMoveAbsoluteDone := TRUE;
END_IF

{warning 'Add method implementation '}
METHOD CalibrateEncValue
END_METHOD

{warning 'Add method implementation '}
METHOD EncSaveRestore
END_METHOD

{warning 'Add property implementation'}
PROPERTY Error : BOOL
GET
END_GET
END_PROPERTY

{warning 'Add property implementation'}
PROPERTY ErrorID : BOOL
GET
END_GET
END_PROPERTY


METHOD FB_Init: BOOL
VAR_INPUT
    bInitRetains: BOOL; // TRUE: the retain variables are initialized (reset warm / reset cold)
    bInCopyCode: BOOL;  // TRUE: the instance will be copied to the copy code afterward (online change)

    AxisReference : REFERENCE TO AXIS_REF;
END_VAR

THIS^.AxisReference REF= AxisReference;
END_METHOD

{warning 'Add method implementation '}
METHOD GearIn
END_METHOD

{warning 'Add method implementation '}
METHOD GearOut
END_METHOD


METHOD GetAxisRef : REFERENCE TO AXIS_REF

GetAxisRef REF= THIS^.AxisReference;
END_METHOD


METHOD GetPowerOverride : LREAL

GetPowerOverride := TO_LREAL(THIS^.AxisReference.PlcToNc.Override) / 10000.0;
END_METHOD


METHOD Halt
VAR_INPUT
    Deceleration	: LREAL := 0.0;
    Jerk	: LREAL := 0.0;
    BufferMode	: MC_BufferMode := .MC_BufferMode.MC_Aborting;
END_VAR
VAR_OUTPUT
    Done	: BOOL;
    Busy	: BOOL;
    Active	: BOOL;
    CommandAborted	: BOOL;
    Error	: BOOL;
    ErrorID	: UDINT;
    ErrorStr	: T_MaxString;
END_VAR

bMostRecentHaltDone := FALSE;

IF NOT HaltBusy THEN
    bCommandedHalt := TRUE;
END_IF

THIS^.fbMcHalt(
    Axis := THIS^.AxisReference,
    Deceleration := Deceleration,
    Jerk := Jerk,
    BufferMode := BufferMode,
    Done => Done,
    Busy => Busy,
    Active => Active,
    CommandAborted => CommandAborted,
    Error => Error,
    ErrorID => ErrorID
);

ErrorStr := '';
END_METHOD


PROPERTY HaltBusy : BOOL
GET

HaltBusy := THIS^.fbMcHalt.Busy;
END_GET
END_PROPERTY


PROPERTY HaltDone : BOOL
GET

HaltDone := THIS^.fbMcHalt.Done OR THIS^.bMostRecentHaltDone;
END_GET
END_PROPERTY


PROPERTY HaltError : BOOL
GET

HaltError := THIS^.fbMcHalt.Error;
END_GET
END_PROPERTY


PROPERTY HaltErrorID : UDINT
GET

HaltErrorID := THIS^.fbMcHalt.ErrorID;
END_GET
END_PROPERTY


METHOD Home
VAR_INPUT
    Position : LREAL := DEFAULT_HOME_POSITION;
    HomingMode : MC_HomingMode := MC_DefaultHoming;
END_VAR
VAR_OUTPUT
    Done	: BOOL;
    Busy	: BOOL;
    Active	: BOOL;
    CommandAborted	: BOOL;
    Error	: BOOL;
    ErrorID	: UDINT;
    ErrorStr	: T_MaxString;
END_VAR

bMostRecentHomeDone := FALSE;

IF NOT HomeBusy THEN
    bCommandedHome := TRUE;
END_IF

THIS^.fbMcHome(
    Axis := THIS^.AxisReference,
    HomingMode := HomingMode,
    Done => Done,
    Busy => Busy,
    Active => Active,
    CommandAborted => CommandAborted,
    Error => Error,
    ErrorID => ErrorID
);

ErrorStr := '';
END_METHOD


PROPERTY HomeBusy : BOOL
GET

HomeBusy := THIS^.fbMcHome.Busy;
END_GET
END_PROPERTY


PROPERTY HomeDone : BOOL
GET

HomeDone := THIS^.fbMcHome.Done;
END_GET
END_PROPERTY


PROPERTY MeasuredAcceleration : LREAL
GET

MeasuredAcceleration := THIS^.AxisReference.NcToPlc.ActAcc;
END_GET
END_PROPERTY


PROPERTY MeasuredPosition : LREAL
GET

MeasuredPosition := THIS^.AxisReference.NcToPlc.ActPos;
END_GET
END_PROPERTY


PROPERTY MeasuredVelocity : LREAL
GET

MeasuredVelocity := THIS^.AxisReference.NcToPlc.ActVelo;
END_GET
END_PROPERTY


METHOD MoveAbsolute
VAR_INPUT
    Position	: LREAL;
    Velocity	: LREAL;
    Acceleration	: LREAL := 0.0;
    Deceleration	: LREAL := 0.0;
    Jerk	: LREAL := 0.0;
    BufferMode	: MC_BufferMode := .MC_BufferMode.MC_Aborting;
END_VAR
VAR_OUTPUT
    Done	: BOOL;
    Busy	: BOOL;
    Active	: BOOL;
    CommandAborted	: BOOL;
    Error	: BOOL;
    ErrorID	: UDINT;
    ErrorStr	: T_MaxString;
END_VAR

bMostRecentMoveAbsoluteDone := FALSE;

IF NOT MoveAbsoluteBusy THEN
    bCommandedMoveAbsolute := TRUE;
END_IF

THIS^.fbMcMoveAbsolute(
    Axis := THIS^.AxisReference,
    Position := Position,
    Velocity := Velocity,
    Acceleration := Acceleration,
    Deceleration := Deceleration,
    Jerk := Jerk,
    BufferMode := BufferMode,
    Done => Done,
    Busy => Busy,
    Active => Active,
    CommandAborted => CommandAborted,
    Error => Error,
    ErrorID => ErrorID
);

ErrorStr := '';
END_METHOD


PROPERTY MoveAbsoluteBusy : BOOL
GET

MoveAbsoluteBusy := THIS^.fbMcMoveAbsolute.Busy;
END_GET
END_PROPERTY


PROPERTY MoveAbsoluteDone : BOOL
GET

MoveAbsoluteDone := THIS^.fbMcMoveAbsolute.Done OR THIS^.bMostRecentMoveAbsoluteDone;
END_GET
END_PROPERTY


PROPERTY MoveAbsoluteError : BOOL
GET

MoveAbsoluteError := THIS^.fbMcMoveAbsolute.Error;
END_GET
END_PROPERTY


PROPERTY MoveAbsoluteErrorID : UDINT
GET

MoveAbsoluteErrorID := THIS^.fbMcMoveAbsolute.ErrorID;
END_GET
END_PROPERTY


PROPERTY MoveAbsoluteTargetAcceleration : LREAL
GET

MoveAbsoluteTargetAcceleration := THIS^.fbMcMoveAbsolute.Acceleration;
END_GET
END_PROPERTY


PROPERTY MoveAbsoluteTargetDeceleration : LREAL
GET

MoveAbsoluteTargetDeceleration := THIS^.fbMcMoveAbsolute.Deceleration;
END_GET
END_PROPERTY


PROPERTY MoveAbsoluteTargetJerk : LREAL
GET

MoveAbsoluteTargetJerk := THIS^.fbMcMoveAbsolute.Jerk;
END_GET
END_PROPERTY


PROPERTY MoveAbsoluteTargetPosition : LREAL
GET

MoveAbsoluteTargetPosition := THIS^.fbMcMoveAbsolute.Position;
END_GET
END_PROPERTY


PROPERTY MoveAbsoluteTargetVelocity : LREAL
GET

MoveAbsoluteTargetVelocity := THIS^.fbMcMoveAbsolute.Velocity;
END_GET
END_PROPERTY


PROPERTY MoveBusy : BOOL
GET

MoveBusy := HaltBusy OR HomeBusy OR MoveAbsoluteBusy;
END_GET
END_PROPERTY


PROPERTY MoveDone : BOOL
GET

MoveDone := HaltDone AND HomeDone AND MoveAbsoluteDone;
END_GET
END_PROPERTY


PROPERTY NegativeMotionIsEnabled : BOOL
GET

NegativeMotionIsEnabled := THIS^.AxisReference.PlcToNc.ControlDWord.2;
END_GET
END_PROPERTY


PROPERTY PositiveMotionIsEnabled : BOOL
GET

PositiveMotionIsEnabled := THIS^.AxisReference.PlcToNc.ControlDWord.1;
END_GET
END_PROPERTY


METHOD Power
VAR_INPUT
    Enable	: BOOL;
    Enable_Positive	: BOOL;
    Enable_Negative	: BOOL;
    (* in percent from 0 to 100 *)
    Override	: LREAL := 100.0;
    BufferMode	: MC_BufferMode := .MC_BufferMode.MC_Aborting;
END_VAR
VAR_OUTPUT
    Status	: BOOL;
    Busy	: BOOL;
    Active	: BOOL;
    Error	: BOOL;
    ErrorID	: UDINT;
    ErrorStr	: T_MaxString;
END_VAR

THIS^.fbMcPower(
    Axis := THIS^.AxisReference,
    Enable := Enable,
    Enable_Positive := Enable_Positive,
    Enable_Negative := Enable_Negative,
    Override := Override,
    BufferMode := BufferMode,
    Status => Status,
    Busy => Busy,
    Active => Active,
    Error => Error,
    ErrorID => ErrorID
);

ErrorStr := '';
END_METHOD


PROPERTY PowerError : BOOL
GET

PowerError := THIS^.fbMcPower.Error;
END_GET
END_PROPERTY


PROPERTY PowerErrorID : UDINT
GET

PowerErrorID := THIS^.fbMcPower.ErrorID;
END_GET
END_PROPERTY


PROPERTY PowerIsEnabled : BOOL
GET

PowerIsEnabled := THIS^.AxisReference.PlcToNc.ControlDWord.0;
END_GET
END_PROPERTY


PROPERTY PowerOverride : LREAL
GET

PowerOverride := GetPowerOverride();
END_GET
END_PROPERTY

{warning 'Add property implementation'}
PROPERTY PowerStatus : BOOL
GET

PowerStatus := THIS^.fbMcPower.Status;
END_GET
END_PROPERTY


METHOD Reset
VAR_OUTPUT
    Done	: BOOL;
    Busy	: BOOL;
    Error	: BOOL;
    ErrorID	: UDINT;
    ErrorStr	: T_MaxString;
END_VAR

bMostRecentResetDone := FALSE;

IF NOT ResetBusy THEN
    bCommandedReset := TRUE;
END_IF

THIS^.fbMcReset(
    Axis := THIS^.AxisReference,
    Done => Done,
    Busy => Busy,
    Error => Error,
    ErrorID => ErrorID,
);

ErrorStr := '';
END_METHOD


PROPERTY ResetBusy : BOOL
GET

ResetBusy := fbMcReset.Busy;
END_GET
END_PROPERTY


PROPERTY ResetDone : BOOL
GET

ResetDone := fbMcReset.Done;
END_GET
END_PROPERTY


PROPERTY ResetError : BOOL
GET

ResetError := fbMcReset.Error;
END_GET
END_PROPERTY


PROPERTY ResetErrorID : UDINT
GET

ResetErrorID := fbMcReset.ErrorID;
END_GET
END_PROPERTY


PROPERTY SetpointAcceleration : LREAL
GET

SetpointAcceleration := THIS^.AxisReference.NcToPlc.SetAcc;
END_GET
END_PROPERTY


PROPERTY SetpointJerk : LREAL
GET

SetpointJerk := THIS^.AxisReference.NcToPlc.SetJerk;
END_GET
END_PROPERTY


PROPERTY SetpointPosition : LREAL
GET

SetpointPosition := THIS^.AxisReference.NcToPlc.SetPos;
END_GET
END_PROPERTY


PROPERTY SetpointVelocity : LREAL
GET

SetpointVelocity := THIS^.AxisReference.NcToPlc.SetVelo;
END_GET
END_PROPERTY


METHOD SetPowerOverride
VAR_INPUT
    (* in percent from 0 to 100 *)
    Override	: LREAL;
END_VAR
VAR_OUTPUT
    Status	: BOOL;
    Busy	: BOOL;
    Active	: BOOL;
    Error	: BOOL;
    ErrorID	: UDINT;
    ErrorStr	: T_MaxString;
END_VAR

THIS^.fbMcPower(
    Axis := THIS^.AxisReference,
    Override := Override,
    Status => Status,
    Busy => Busy,
    Error => Error,
    ErrorID => ErrorID
);

ErrorStr := '';
END_METHOD

END_FUNCTION_BLOCK

// ---- POUs/Motion/FB_MotionAxisNCContinuous.TcPOU

FUNCTION_BLOCK FB_MotionAxisNCContinuous EXTENDS FB_MotionAxisNC IMPLEMENTS I_MotionAxisContinuous
VAR
    bCommandedMoveVelocity1 : BOOL;
    bCommandedMoveVelocity2 : BOOL;
    fbMcMoveVelocity1 : MC_MoveVelocity;
    fbMcMoveVelocity2 : MC_MoveVelocity;
    eMotionDirection : MC_Direction := MC_Direction.MC_Undefined_Direction;
    fTargetPosition : LREAL;
END_VAR


SUPER^();

THIS^.fbMcMoveVelocity1(
    Axis := THIS^.AxisReference,
    Execute := THIS^.bCommandedMoveVelocity1
);
THIS^.bCommandedMoveVelocity1 := FALSE;

THIS^.fbMcMoveVelocity2(
    Axis := THIS^.AxisReference,
    Execute := THIS^.bCommandedMoveVelocity2
);
THIS^.bCommandedMoveVelocity2 := FALSE;


PROPERTY MoveBusy : BOOL
GET

MoveBusy := SUPER^.MoveBusy OR THIS^.MoveContinuousBusy;
END_GET
END_PROPERTY


METHOD MoveContinuous
VAR_INPUT
    Position	: LREAL;
    Velocity	: LREAL;
    Acceleration	: LREAL := 0.0;
    Deceleration	: LREAL := 0.0;
    Jerk	: LREAL := 0.0;
    BufferMode	: MC_BufferMode := .MC_BufferMode.MC_Aborting;
END_VAR
VAR_OUTPUT
    InVelocity	: BOOL;
    Busy	: BOOL;
    Active	: BOOL;
    CommandAborted	: BOOL;
    Error	: BOOL;
    ErrorID	: UDINT;
    ErrorStr	: T_MaxString;
END_VAR

IF Position > THIS^.MeasuredPosition THEN
    THIS^.eMotionDirection := MC_Direction.MC_Positive_Direction;
ELSIF Position < THIS^.MeasuredPosition THEN
    THIS^.eMotionDirection := MC_Direction.MC_Negative_Direction;
ELSE
    RETURN;
END_IF

THIS^.fTargetPosition := Position;

IF NOT fbMcMoveVelocity1.Busy THEN
    THIS^.bCommandedMoveVelocity1 := TRUE;
    THIS^.fbMcMoveVelocity1(
        Axis := THIS^.AxisReference,
        Velocity := Velocity,
        Acceleration := Acceleration,
        Deceleration := Deceleration,
        Jerk := Jerk,
        Direction := THIS^.eMotionDirection,
        BufferMode := BufferMode,
        InVelocity => InVelocity,
        Busy => Busy,
        Active => Active,
        CommandAborted => CommandAborted,
        Error => Error,
        ErrorID => ErrorID
    );
ELSE
    THIS^.bCommandedMoveVelocity2 := TRUE;
    THIS^.fbMcMoveVelocity2(
        Axis := THIS^.AxisReference,
        Velocity := Velocity,
        Acceleration := Acceleration,
        Deceleration := Deceleration,
        Jerk := Jerk,
        Direction := THIS^.eMotionDirection,
        BufferMode := BufferMode,
        InVelocity => InVelocity,
        Busy => Busy,
        Active => Active,
        CommandAborted => CommandAborted,
        Error => Error,
        ErrorID => ErrorID
    );
END_IF

ErrorStr := '';
END_METHOD


PROPERTY MoveContinuousBusy : BOOL
GET

MoveContinuousBusy := THIS^.fbMcMoveVelocity1.Busy OR THIS^.fbMcMoveVelocity2.Busy;
END_GET
END_PROPERTY


PROPERTY MoveContinuousError : BOOL
GET

MoveContinuousError := THIS^.fbMcMoveVelocity1.Error OR THIS^.fbMcMoveVelocity2.Error;
END_GET
END_PROPERTY


PROPERTY MoveContinuousErrorID : UDINT
GET

IF THIS^.fbMcMoveVelocity1.ErrorID <> 0 THEN
    MoveContinuousErrorID := THIS^.fbMcMoveVelocity1.ErrorID;
ELSE
    MoveContinuousErrorID := THIS^.fbMcMoveVelocity2.ErrorID;
END_IF
END_GET
END_PROPERTY


PROPERTY MoveContinuousInVelocity : BOOL
GET

MoveContinuousInVelocity := THIS^.fbMcMoveVelocity1.InVelocity OR THIS^.fbMcMoveVelocity2.InVelocity;
END_GET
END_PROPERTY

PROPERTY MoveContinuousPassedTargetPosition : BOOL
GET

CASE THIS^.eMotionDirection OF
    MC_Direction.MC_Positive_Direction :
        MoveContinuousPassedTargetPosition := THIS^.fTargetPosition <= THIS^.MeasuredPosition;

    MC_Direction.MC_Negative_Direction :
        MoveContinuousPassedTargetPosition := THIS^.fTargetPosition >= THIS^.MeasuredPosition;

    MC_Direction.MC_Undefined_Direction :
        MoveContinuousPassedTargetPosition := THIS^.fTargetPosition = THIS^.MeasuredPosition;;
END_CASE
END_GET
END_PROPERTY


PROPERTY MoveDone : BOOL
GET

MoveDone := SUPER^.MoveDone AND THIS^.MoveContinuousPassedTargetPosition AND THIS^.MoveContinuousInVelocity;
END_GET
END_PROPERTY

END_FUNCTION_BLOCK

// ---- POUs/Motion/FB_MotionAxisPneumatic.TcPOU
FUNCTION_BLOCK FB_MotionAxisPneumatic IMPLEMENTS I_MotionAxis
VAR_INPUT
END_VAR
VAR_OUTPUT
END_VAR
VAR
END_VAR

{warning 'Add method implementation '}
METHOD CalibrateEncValue
END_METHOD

{warning 'Add method implementation '}
METHOD EncSaveRestore
END_METHOD

{warning 'Add property implementation'}
PROPERTY Error : BOOL
GET
END_GET
END_PROPERTY

{warning 'Add property implementation'}
PROPERTY ErrorID : BOOL
GET
END_GET
END_PROPERTY

{warning 'Add method implementation '}
METHOD GearIn
END_METHOD

{warning 'Add method implementation '}
METHOD GearOut
END_METHOD

{warning 'Add method implementation '}
METHOD GetAxisRef : REFERENCE TO AXIS_REF
END_METHOD

{warning 'Add method implementation '}
METHOD GetPowerOverride : LREAL
END_METHOD

{warning 'Add method implementation '}
METHOD Halt
VAR_INPUT
    Deceleration	: LREAL := 0.0;
    Jerk	: LREAL := 0.0;
    BufferMode	: MC_BufferMode := .MC_BufferMode.MC_Aborting;
END_VAR
VAR_OUTPUT
    Done	: BOOL;
    Busy	: BOOL;
    Active	: BOOL;
    CommandAborted	: BOOL;
    Error	: BOOL;
    ErrorID	: UDINT;
    ErrorStr	: T_MaxString;
END_VAR
END_METHOD

{warning 'Add property implementation'}
PROPERTY HaltBusy : BOOL
GET
END_GET
END_PROPERTY

{warning 'Add property implementation'}
PROPERTY HaltDone : BOOL
GET
END_GET
END_PROPERTY

{warning 'Add property implementation'}
PROPERTY HaltError : BOOL
GET
END_GET
END_PROPERTY

{warning 'Add property implementation'}
PROPERTY HaltErrorID : UDINT
GET
END_GET
END_PROPERTY

{warning 'Add method implementation '}
METHOD Home
VAR_INPUT
    Position : LREAL := DEFAULT_HOME_POSITION;
    HomingMode : MC_HomingMode := MC_DefaultHoming;
END_VAR
VAR_OUTPUT
    Done	: BOOL;
    Busy	: BOOL;
    Active	: BOOL;
    CommandAborted	: BOOL;
    Error	: BOOL;
    ErrorID	: UDINT;
    ErrorStr	: T_MaxString;
END_VAR
END_METHOD

{warning 'Add property implementation'}
PROPERTY HomeBusy : BOOL
GET
END_GET
END_PROPERTY

{warning 'Add property implementation'}
PROPERTY HomeDone : BOOL
GET
END_GET
END_PROPERTY

{warning 'Add property implementation'}
PROPERTY MeasuredAcceleration : LREAL
GET
END_GET
END_PROPERTY

{warning 'Add property implementation'}
PROPERTY MeasuredPosition : LREAL
GET
END_GET
END_PROPERTY

{warning 'Add property implementation'}
PROPERTY MeasuredVelocity : LREAL
GET
END_GET
END_PROPERTY

{warning 'Add method implementation '}
METHOD MoveAbsolute
VAR_INPUT
    Position	: LREAL;
    Velocity	: LREAL;
    Acceleration	: LREAL := 0.0;
    Deceleration	: LREAL := 0.0;
    Jerk	: LREAL := 0.0;
    BufferMode	: MC_BufferMode := .MC_BufferMode.MC_Aborting;
END_VAR
VAR_OUTPUT
    Done	: BOOL;
    Busy	: BOOL;
    Active	: BOOL;
    CommandAborted	: BOOL;
    Error	: BOOL;
    ErrorID	: UDINT;
    ErrorStr	: T_MaxString;
END_VAR
END_METHOD

{warning 'Add property implementation'}
PROPERTY MoveAbsoluteBusy : BOOL
GET
END_GET
END_PROPERTY

{warning 'Add property implementation'}
PROPERTY MoveAbsoluteDone : BOOL
GET
END_GET
END_PROPERTY

{warning 'Add property implementation'}
PROPERTY MoveAbsoluteError : BOOL
GET
END_GET
END_PROPERTY

{warning 'Add property implementation'}
PROPERTY MoveAbsoluteErrorID : UDINT
GET
END_GET
END_PROPERTY

{warning 'Add property implementation'}
PROPERTY MoveAbsoluteTargetAcceleration : LREAL
GET
END_GET
END_PROPERTY

{warning 'Add property implementation'}
PROPERTY MoveAbsoluteTargetDeceleration : LREAL
GET
END_GET
END_PROPERTY

{warning 'Add property implementation'}
PROPERTY MoveAbsoluteTargetJerk : LREAL
GET
END_GET
END_PROPERTY

{warning 'Add property implementation'}
PROPERTY MoveAbsoluteTargetPosition : LREAL
GET
END_GET
END_PROPERTY

{warning 'Add property implementation'}
PROPERTY MoveAbsoluteTargetVelocity : LREAL
GET
END_GET
END_PROPERTY

{warning 'Add property implementation'}
PROPERTY MoveBusy : BOOL
GET
END_GET
END_PROPERTY

{warning 'Add property implementation'}
PROPERTY MoveDone : BOOL
GET
END_GET
END_PROPERTY

{warning 'Add property implementation'}
PROPERTY NegativeMotionIsEnabled : BOOL
GET
END_GET
END_PROPERTY

{warning 'Add property implementation'}
PROPERTY PositiveMotionIsEnabled : BOOL
GET
END_GET
END_PROPERTY

{warning 'Add method implementation '}
METHOD Power
VAR_INPUT
    Enable	: BOOL;
    Enable_Positive	: BOOL;
    Enable_Negative	: BOOL;
    (* in percent from 0 to 100 *)
    Override	: LREAL := 100.0;
    BufferMode	: MC_BufferMode := .MC_BufferMode.MC_Aborting;
END_VAR
VAR_OUTPUT
    Status	: BOOL;
    Busy	: BOOL;
    Active	: BOOL;
    Error	: BOOL;
    ErrorID	: UDINT;
    ErrorStr	: T_MaxString;
END_VAR
END_METHOD

{warning 'Add property implementation'}
PROPERTY PowerError : BOOL
GET
END_GET
END_PROPERTY

{warning 'Add property implementation'}
PROPERTY PowerErrorID : UDINT
GET
END_GET
END_PROPERTY

{warning 'Add property implementation'}
PROPERTY PowerIsEnabled : BOOL
GET
END_GET
END_PROPERTY

{warning 'Add property implementation'}
PROPERTY PowerOverride : LREAL
GET
END_GET
END_PROPERTY

{warning 'Add property implementation'}
PROPERTY PowerStatus : BOOL
GET
END_GET
END_PROPERTY

{warning 'Add method implementation '}
METHOD Reset
VAR_OUTPUT
    Done	: BOOL;
    Busy	: BOOL;
    Error	: BOOL;
    ErrorID	: UDINT;
    ErrorStr	: T_MaxString;
END_VAR
END_METHOD

{warning 'Add property implementation'}
PROPERTY ResetBusy : BOOL
GET
END_GET
END_PROPERTY

{warning 'Add property implementation'}
PROPERTY ResetDone : BOOL
GET
END_GET
END_PROPERTY

{warning 'Add property implementation'}
PROPERTY ResetError : BOOL
GET
END_GET
END_PROPERTY

{warning 'Add property implementation'}
PROPERTY ResetErrorID : UDINT
GET
END_GET
END_PROPERTY

{warning 'Add property implementation'}
PROPERTY SetpointAcceleration : LREAL
GET
END_GET
END_PROPERTY

{warning 'Add property implementation'}
PROPERTY SetpointJerk : LREAL
GET
END_GET
END_PROPERTY

{warning 'Add property implementation'}
PROPERTY SetpointPosition : LREAL
GET
END_GET
END_PROPERTY

{warning 'Add property implementation'}
PROPERTY SetpointVelocity : LREAL
GET
END_GET
END_PROPERTY

{warning 'Add method implementation '}
METHOD SetPowerOverride
VAR_INPUT
    (* in percent from 0 to 100 *)
    Override	: LREAL;
END_VAR
VAR_OUTPUT
    Status	: BOOL;
    Busy	: BOOL;
    Active	: BOOL;
    Error	: BOOL;
    ErrorID	: UDINT;
    ErrorStr	: T_MaxString;
END_VAR
END_METHOD

END_FUNCTION_BLOCK

// ---- POUs/Motion/States/FB_PositionStateMoveND.TcPOU

FUNCTION_BLOCK FB_PositionStateMoveND
(*
    This function block coordinates multidimensional state moves for groups of motors.
    It is a building block not meant for use outside of lcls-twintcat-motion.

    Use FB_PositionState1D, FB_PositionState2D, ... etc. instead
*)
VAR_IN_OUT
    // Array of motors to move together
    astMotionStage: ARRAY[1..MotionConstants.MAX_STATE_MOTORS] OF ST_MotionStage;
    // 1D Position states: the current position to send each axis to
    astPositionState: ARRAY[1..MotionConstants.MAX_STATE_MOTORS] OF ST_PositionState;
END_VAR
VAR_INPUT
    // The number of motors we're actually using
    nActiveMotorCount: UINT;
    // Start all moves on rising edge, stop all moves on falling edge
    bExecute: BOOL;
    // Reset any errors
    bReset: BOOL;
    // Define behavior for when a move request is interrupted with a new request
    enumMotionRequest: E_MotionRequest := E_MotionRequest.WAIT;
END_VAR
VAR_OUTPUT
    // TRUE if ALL of the motors are at their goal states
    bAtState: BOOL;
    // TRUE if ANY of this FB's moves are in progress
    bBusy: BOOL;
    // TRUE if ALL motors have completed the last move request from this FB
    bDone: BOOL;
    // TRUE if ANY of this FB's moves had an error
    bError: BOOL;
    // How many FBs are erroring
    nErrorCount: UINT;
    // Which component is the source of the example/summarized error
    nShownError: DINT;
    // One of the error ids
    nErrorID: UDINT;
    // The error error message matching the ID
    sErrorMessage: STRING;
END_VAR
VAR
    // 1D State movers: FBs to move the motors
    afbPositionStateMove: ARRAY[1..MotionConstants.MAX_STATE_MOTORS] OF FB_PositionStateMove;
    nIndex: DINT;
    bMotorCountError: BOOL;
    nLowerBound: DINT;
    nUpperBound: DINT;
    rtExec: R_TRIG;
    nNextMove: DINT;
END_VAR


rtExec(CLK:=bExecute);

CheckCount();
IF NOT bMotorCountError THEN
    DoStateMoves();
    CombineOutputs();
END_IF

ACTION CheckCount:

// Make sure the motor count is valid (positive, nonzero, less or equal to the max)
bMotorCountError S= nActiveMotorCount <= 0;
bMotorCountError S= nActiveMotorCount > MotionConstants.MAX_STATE_MOTORS;

IF bMotorCountError THEN
    bError := TRUE;
    sErrorMessage := 'Internal Error: invalid motor count';
END_IF
END_ACTION

ACTION CombineOutputs:

// bAtState is TRUE if ALL entries are TRUE
bAtState := TRUE;
FOR nIndex := 1 TO nActiveMotorCount DO
    bAtState := bAtState AND afbPositionStateMove[nIndex].bAtState;
END_FOR

// bBusy is TRUE if ANY entry is TRUE
bBusy := FALSE;
FOR nIndex := 1 TO nActiveMotorCount DO
    bBusy := bBusy OR afbPositionStateMove[nIndex].bBusy;
END_FOR

// bDone is TRUE if ALL entries are TRUE
bDone := TRUE;
FOR nIndex := 1 TO nActiveMotorCount DO
    bDone := bDone AND afbPositionStateMove[nIndex].bDone;
END_FOR

// bError is TRUE if ANY entry is TRUE
// also set nShownError and increment nErrorCount
bError := FALSE;
nErrorCount := 0;
FOR nIndex := 1 TO nActiveMotorCount DO
    bError := bError OR afbPositionStateMove[nIndex].bError;
    IF afbPositionStateMove[nIndex].bError THEN
        nShownError := nIndex;
        nErrorCount := nErrorCount + 1;
    END_IF
END_FOR

// Pick error id and message using nShownError
IF bError THEN
    nErrorID := afbPositionStateMove[nShownError].nErrorID;
    sErrorMessage := afbPositionStateMove[nShownError].sErrorMessage;
ELSE
    nErrorID := 0;
    sErrorMessage := '';
END_IF
END_ACTION

ACTION DoStateMoves:

// Do the individual moves
IF rtExec.Q THEN
    FOR nIndex := 1 TO nActiveMotorCount DO
        astPositionState[nIndex].bMoveQueued := rtExec.Q;
    END_FOR
END_IF

FOR nIndex := 1 TO nActiveMotorCount DO
    IF bError OR bReset OR astMotionStage[nIndex].bBusy OR astMotionStage[nIndex].bDone THEN
        astPositionState[nIndex].bMoveQueued := FALSE;
    END_IF
END_FOR

nNextMove := nActiveMotorCount + 1;
FOR nIndex := 1 TO nActiveMotorCount DO
    IF astPositionState[nIndex].bMoveQueued AND astPositionState[nIndex].nMoveOrder < nNextMove THEN
        nNextMove := astPositionState[nIndex].nMoveOrder;
    END_IF
END_FOR

FOR nIndex := 1 TO nActiveMotorCount DO
    afbPositionStateMove[nIndex](
        stMotionStage:=astMotionStage[nIndex],
        stPositionState:=astPositionState[nIndex],
        bExecute:=astPositionState[nIndex].bMoveQueued AND astPositionState[nIndex].nMoveOrder = nNextMove,
        bReset:=bReset,
        enumMotionRequest:=enumMotionRequest,
    );
END_FOR
END_ACTION

END_FUNCTION_BLOCK

// ---- Tests/FB_MotionAxisNC_Test.TcPOU

FUNCTION_BLOCK FB_MotionAxisNC_Test EXTENDS FB_TestSuite
VAR
    AxisReference : AXIS_REF;
END_VAR


GivenLinkedAxisRefExpectSequenceOfOperationsSuccessful();


METHOD PRIVATE GivenLinkedAxisRefExpectSequenceOfOperationsSuccessful
VAR_INST
    nTestStep : INT;
    fbTestTimer : TON := (PT := T#10s);

    fbMotionAxisNC : FB_MotionAxisNC(
        AxisReference := THIS^.AxisReference
    );
END_VAR

TEST(__POUNAME());

fbTestTimer(IN := TRUE);

fbMotionAxisNC();

CASE nTestStep OF
    0:
        fbMotionAxisNC.Reset();
        fbMotionAxisNC.Power(
            Enable := FALSE,
            Enable_Positive := FALSE,
            Enable_Negative := FALSE
        );

        nTestStep := nTestStep + 1;
    1:
        IF fbMotionAxisNC.ResetDone AND
            NOT fbMotionAxisNC.PowerIsEnabled AND
            NOT fbMotionAxisNC.PositiveMotionIsEnabled AND
            NOT fbMotionAxisNC.NegativeMotionIsEnabled THEN
            AssertFalse(
                Condition := fbMotionAxisNC.PowerError,
                Message := 'Move should not show an error.'
            );
            AssertEquals_UDINT(
                Expected := 0,
                Actual := fbMotionAxisNC.PowerErrorID,
                Message := 'Error ID should be 0.'
            );

            AssertFalse(
                Condition := fbMotionAxisNC.MoveAbsoluteBusy,
                Message := 'Move should not show as busy.'
            );
            AssertFalse(
                Condition := fbMotionAxisNC.MoveAbsoluteDone,
                Message := 'Move should not show as done.'
            );
            AssertFalse(
                Condition := fbMotionAxisNC.MoveAbsoluteError,
                Message := 'Move should not show an error.'
            );
            AssertEquals_UDINT(
                Expected := 0,
                Actual := fbMotionAxisNC.MoveAbsoluteErrorID,
                Message := 'Error ID should be 0.'
            );

            nTestStep := nTestStep + 1;
        END_IF
    2:
        fbMotionAxisNC.Power(
            Enable := TRUE,
            Enable_Positive := TRUE,
            Enable_Negative := TRUE,
            Override := 90.0
        );

        nTestStep := nTestStep + 1;
    3:
        IF fbMotionAxisNC.PowerIsEnabled AND
            fbMotionAxisNC.PositiveMotionIsEnabled AND
            fbMotionAxisNC.NegativeMotionIsEnabled THEN
            AssertEquals_LREAL(
                Expected := 90.0,
                Actual := fbMotionAxisNC.GetPowerOverride(),
                Delta := 0.0,
                Message := 'GetPowerOverride() did not return the expected value.'
            );
            AssertEquals_LREAL(
                Expected := 90.0,
                Actual := fbMotionAxisNC.PowerOverride,
                Delta := 0.0,
                Message := 'PowerOverride was not the expected value.'
            );
            AssertFalse(
                Condition := fbMotionAxisNC.PowerError,
                Message := 'Move should not show an error.'
            );
            AssertEquals_UDINT(
                Expected := 0,
                Actual := fbMotionAxisNC.PowerErrorID,
                Message := 'Error ID should be 0.'
            );

            nTestStep := nTestStep + 1;
        END_IF
    4:
        fbMotionAxisNC.MoveAbsolute(
            Position := 15.0,
            Velocity := 16.0,
            Acceleration := 17.0,
            Deceleration := 18.0,
            Jerk := 19.0,
            BufferMode := MC_BufferMode.MC_BlendingHigh
        );

        nTestStep := nTestStep + 1;
    5:
         IF fbMotionAxisNC.MoveAbsoluteBusy THEN
            AssertFalse(
                Condition := fbMotionAxisNC.MoveAbsoluteDone,
                Message := 'Move should not show as done.'
            );
            AssertEquals_LREAL(
                Expected := 15.0,
                Actual := fbMotionAxisNC.MoveAbsoluteTargetPosition,
                Delta := 0.0,
                Message := 'Position setpoint was not the expected value.'
            );
            AssertEquals_LREAL(
                Expected := 16.0,
                Actual := fbMotionAxisNC.MoveAbsoluteTargetVelocity,
                Delta := 0.0,
                Message := 'Velocity setpoint was not the expected value.'
            );
            AssertEquals_LREAL(
                Expected := 17.0,
                Actual := fbMotionAxisNC.MoveAbsoluteTargetAcceleration,
                Delta := 0.0,
                Message := 'Acceleration setpoint was not the expected value.'
            );
            AssertEquals_LREAL(
                Expected := 18.0,
                Actual := fbMotionAxisNC.MoveAbsoluteTargetDeceleration,
                Delta := 0.0,
                Message := 'Deceleration setpoint was not the expected value.'
            );
            AssertEquals_LREAL(
                Expected := 19.0,
                Actual := fbMotionAxisNC.MoveAbsoluteTargetJerk,
                Delta := 0.0,
                Message := 'Jerk setpoint was not the expected value.'
            );
            AssertFalse(
                Condition := fbMotionAxisNC.MoveAbsoluteError,
                Message := 'Move should not show an error.'
            );
            AssertEquals_UDINT(
                Expected := 0,
                Actual := fbMotionAxisNC.MoveAbsoluteErrorID,
                Message := 'Error ID should be 0.'
            );

            nTestStep := nTestStep + 1;
        END_IF
    6:
         IF fbMotionAxisNC.MoveAbsoluteDone THEN
            AssertFalse(
                Condition := fbMotionAxisNC.MoveAbsoluteBusy,
                Message := 'Move should not show as busy.'
            );
            AssertEquals_LREAL(
                Expected := 15.0,
                Actual := fbMotionAxisNC.MeasuredPosition,
                Delta := 1e-3,
                Message := 'Measured position was not the expected value.'
            );
            AssertEquals_LREAL(
                Expected := 0.0,
                Actual := fbMotionAxisNC.MeasuredVelocity,
                Delta := 1.0,
                Message := 'Measured velocity was not the expected value.'
            );
            AssertEquals_LREAL(
                Expected := 0.0,
                Actual := fbMotionAxisNC.MeasuredAcceleration,
                Delta := 1.0,
                Message := 'Measured acceleration was not the expected value.'
            );
            AssertFalse(
                Condition := fbMotionAxisNC.MoveAbsoluteError,
                Message := 'Move should not show an error.'
            );
            AssertEquals_UDINT(
                Expected := 0,
                Actual := fbMotionAxisNC.MoveAbsoluteErrorID,
                Message := 'Error ID should be 0.'
            );

            nTestStep := nTestStep + 1;
        END_IF
    7:
        fbMotionAxisNC.MoveAbsolute(
            Position := 16.0,
            Velocity := 17.0,
            Acceleration := 18.0,
            Deceleration := 19.0,
            Jerk := 110.0,
            BufferMode := MC_BufferMode.MC_BlendingHigh
        );

        nTestStep := nTestStep + 1;
    8:
         IF fbMotionAxisNC.MoveAbsoluteBusy THEN
            AssertFalse(
                Condition := fbMotionAxisNC.MoveAbsoluteDone,
                Message := 'Move should not show as done.'
            );
            AssertEquals_LREAL(
                Expected := 16.0,
                Actual := fbMotionAxisNC.MoveAbsoluteTargetPosition,
                Delta := 0.0,
                Message := 'Position setpoint was not the expected value.'
            );
            AssertEquals_LREAL(
                Expected := 17.0,
                Actual := fbMotionAxisNC.MoveAbsoluteTargetVelocity,
                Delta := 0.0,
                Message := 'Velocity setpoint was not the expected value.'
            );
            AssertEquals_LREAL(
                Expected := 18.0,
                Actual := fbMotionAxisNC.MoveAbsoluteTargetAcceleration,
                Delta := 0.0,
                Message := 'Acceleration setpoint was not the expected value.'
            );
            AssertEquals_LREAL(
                Expected := 19.0,
                Actual := fbMotionAxisNC.MoveAbsoluteTargetDeceleration,
                Delta := 0.0,
                Message := 'Deceleration setpoint was not the expected value.'
            );
            AssertEquals_LREAL(
                Expected := 110.0,
                Actual := fbMotionAxisNC.MoveAbsoluteTargetJerk,
                Delta := 0.0,
                Message := 'Jerk setpoint was not the expected value.'
            );
            AssertFalse(
                Condition := fbMotionAxisNC.MoveAbsoluteError,
                Message := 'Move should not show an error.'
            );
            AssertEquals_UDINT(
                Expected := 0,
                Actual := fbMotionAxisNC.MoveAbsoluteErrorID,
                Message := 'Error ID should be 0.'
            );

            nTestStep := nTestStep + 1;
        END_IF
    9:
         IF fbMotionAxisNC.MoveAbsoluteDone THEN
            AssertFalse(
                Condition := fbMotionAxisNC.MoveAbsoluteBusy,
                Message := 'Move should not show as busy.'
            );
            AssertEquals_LREAL(
                Expected := 16.0,
                Actual := fbMotionAxisNC.MeasuredPosition,
                Delta := 1e-3,
                Message := 'Measured position was not the expected value.'
            );
            AssertEquals_LREAL(
                Expected := 0.0,
                Actual := fbMotionAxisNC.MeasuredVelocity,
                Delta := 1.0,
                Message := 'Measured velocity was not the expected value.'
            );
            AssertEquals_LREAL(
                Expected := 0.0,
                Actual := fbMotionAxisNC.MeasuredAcceleration,
                Delta := 1.0,
                Message := 'Measured acceleration was not the expected value.'
            );
            AssertFalse(
                Condition := fbMotionAxisNC.MoveAbsoluteError,
                Message := 'Move should not show an error.'
            );
            AssertEquals_UDINT(
                Expected := 0,
                Actual := fbMotionAxisNC.MoveAbsoluteErrorID,
                Message := 'Error ID should be 0.'
            );

            nTestStep := nTestStep + 1;
        END_IF
    10:
        fbMotionAxisNC.MoveAbsolute(
            Position := 0.0,
            Velocity := 17.0,
            Acceleration := 18.0,
            Deceleration := 19.0,
            Jerk := 110.0,
            BufferMode := MC_BufferMode.MC_BlendingHigh
        );

        nTestStep := nTestStep + 1;
    11:
         IF fbMotionAxisNC.MoveAbsoluteDone THEN
            AssertFalse(
                Condition := fbMotionAxisNC.MoveAbsoluteBusy,
                Message := 'Move should not show as busy.'
            );
            AssertEquals_LREAL(
                Expected := 0.0,
                Actual := fbMotionAxisNC.MeasuredPosition,
                Delta := 1e-3,
                Message := 'Measured position was not the expected value.'
            );
            AssertEquals_LREAL(
                Expected := 0.0,
                Actual := fbMotionAxisNC.MeasuredVelocity,
                Delta := 1.0,
                Message := 'Measured velocity was not the expected value.'
            );
            AssertEquals_LREAL(
                Expected := 0.0,
                Actual := fbMotionAxisNC.MeasuredAcceleration,
                Delta := 1.0,
                Message := 'Measured acceleration was not the expected value.'
            );
            AssertFalse(
                Condition := fbMotionAxisNC.MoveAbsoluteError,
                Message := 'Move should not show an error.'
            );
            AssertEquals_UDINT(
                Expected := 0,
                Actual := fbMotionAxisNC.MoveAbsoluteErrorID,
                Message := 'Error ID should be 0.'
            );

            nTestStep := nTestStep + 1;
        END_IF
    12:
        fbMotionAxisNC.Power(
            Enable := FALSE,
            Enable_Positive := FALSE,
            Enable_Negative := FALSE
        );

        nTestStep := nTestStep + 1;
    13:
        IF NOT fbMotionAxisNC.PowerStatus THEN
            AssertFalse(
                Condition := fbMotionAxisNC.PowerIsEnabled,
                Message := 'Axis should not be enabled.'
            );
            AssertFalse(
                Condition := fbMotionAxisNC.PositiveMotionIsEnabled,
                Message := 'Axis positive motion should not be enabled.'
            );
            AssertFalse(
                Condition := fbMotionAxisNC.NegativeMotionIsEnabled,
                Message := 'Axis negative motion should not be enabled.'
            );

            nTestStep := nTestStep + 1;
        END_IF

END_CASE

IF nTestStep = 14 THEN
    TEST_FINISHED();
ELSIF fbTestTimer.Q THEN
    AssertTrue(
        Condition := FALSE,
        Message := CONCAT('Timed out at step: ', TO_STRING(nTestStep))
    );

    TEST_FINISHED();
END_IF
END_METHOD

END_FUNCTION_BLOCK

// ---- Tests/FB_MotionAxisNCContinuous_Test.TcPOU

FUNCTION_BLOCK FB_MotionAxisNCContinuous_Test EXTENDS FB_TestSuite
VAR
    AxisReference : AXIS_REF;
END_VAR


GivenLinkedAxisRefExpectSequenceOfOperationsSuccessful();


METHOD PRIVATE GivenLinkedAxisRefExpectSequenceOfOperationsSuccessful
VAR_INST
    nTestStep : INT;
    fbTestTimer : TON := (PT := T#10s);

    fbMotionAxisNCContinuous : FB_MotionAxisNCContinuous(
        AxisReference := THIS^.AxisReference
    );
END_VAR

TEST(__POUNAME());

fbTestTimer(IN := TRUE);

fbMotionAxisNCContinuous();

CASE nTestStep OF
    0:
        fbMotionAxisNCContinuous.Reset();

        nTestStep := nTestStep + 1;
    1:
        IF fbMotionAxisNCContinuous.ResetDone THEN
            AssertFalse(
                Condition := fbMotionAxisNCContinuous.PowerError,
                Message := 'Move should not show an error.'
            );
            AssertEquals_UDINT(
                Expected := 0,
                Actual := fbMotionAxisNCContinuous.PowerErrorID,
                Message := 'Error ID should be 0.'
            );

            AssertFalse(
                Condition := fbMotionAxisNCContinuous.MoveContinuousBusy,
                Message := 'Move should not show as busy.'
            );
            AssertFalse(
                Condition := fbMotionAxisNCContinuous.MoveContinuousInVelocity,
                Message := 'Move should not show as done.'
            );
            AssertFalse(
                Condition := fbMotionAxisNCContinuous.MoveContinuousError,
                Message := 'Move should not show an error.'
            );
            AssertEquals_UDINT(
                Expected := 0,
                Actual := fbMotionAxisNCContinuous.MoveContinuousErrorID,
                Message := 'Error ID should be 0.'
            );

            nTestStep := nTestStep + 1;
        END_IF
    2:
        fbMotionAxisNCContinuous.Power(
            Enable := TRUE,
            Enable_Positive := TRUE,
            Enable_Negative := TRUE,
            Override := 100.0
        );

        nTestStep := nTestStep + 1;
    3:
        IF fbMotionAxisNCContinuous.PowerIsEnabled AND
            fbMotionAxisNCContinuous.PositiveMotionIsEnabled AND
            fbMotionAxisNCContinuous.NegativeMotionIsEnabled THEN

            nTestStep := nTestStep + 1;
        END_IF
    4:
        fbMotionAxisNCContinuous.MoveContinuous(
            Position := 50.0,
            Velocity := 25.0,
            Acceleration := 100.0,
            Deceleration := 100.0,
            Jerk := 1000.0,
            BufferMode := MC_BufferMode.MC_Aborting
        );

        nTestStep := nTestStep + 1;
    5:
         IF fbMotionAxisNCContinuous.MoveContinuousBusy THEN
            AssertFalse(
                Condition := fbMotionAxisNCContinuous.MoveContinuousError,
                Message := 'Move should not show an error.'
            );
            AssertEquals_UDINT(
                Expected := 0,
                Actual := fbMotionAxisNCContinuous.MoveContinuousErrorID,
                Message := 'Error ID should be 0.'
            );

            nTestStep := nTestStep + 1;
        END_IF
    6:
         IF fbMotionAxisNCContinuous.MeasuredPosition >= 25.0 THEN
            fbMotionAxisNCContinuous.MoveContinuous(
                Position := -20.0,
                Velocity := 25.0,
                Acceleration := 100.0,
                Deceleration := 100.0,
                Jerk := 1000.0,
                BufferMode := MC_BufferMode.MC_Aborting
            );

            nTestStep := nTestStep + 1;
        END_IF
    7:
         IF fbMotionAxisNCContinuous.MoveContinuousBusy THEN
            AssertFalse(
                Condition := fbMotionAxisNCContinuous.MoveContinuousError,
                Message := 'Move should not show an error.'
            );
            AssertEquals_UDINT(
                Expected := 0,
                Actual := fbMotionAxisNCContinuous.MoveContinuousErrorID,
                Message := 'Error ID should be 0.'
            );

            nTestStep := nTestStep + 1;
        END_IF
    8:
         IF fbMotionAxisNCContinuous.MeasuredPosition <= -5.0 THEN
            fbMotionAxisNCContinuous.MoveAbsolute(
                Position := 0.0,
                Velocity := 12.0,
                Acceleration := 113.0,
                Deceleration := 100.0,
                Jerk := 1540.0,
                BufferMode := MC_BufferMode.MC_Aborting
            );

            nTestStep := nTestStep + 1;
        END_IF

         IF fbMotionAxisNCContinuous.MoveAbsoluteBusy THEN
            nTestStep := nTestStep + 1;
        END_IF
    9:
         IF fbMotionAxisNCContinuous.MoveAbsoluteDone THEN
            AssertEquals_LREAL(
                Expected := 0.0,
                Actual := fbMotionAxisNCContinuous.MeasuredPosition,
                Delta := 1e-3,
                Message := 'Measured position was not the expected value.'
            );
            AssertFalse(
                Condition := fbMotionAxisNCContinuous.MoveAbsoluteError,
                Message := 'Move should not show an error.'
            );
            AssertEquals_UDINT(
                Expected := 0,
                Actual := fbMotionAxisNCContinuous.MoveAbsoluteErrorID,
                Message := 'Error ID should be 0.'
            );

            nTestStep := nTestStep + 1;
        END_IF
    10:
        fbMotionAxisNCContinuous.Power(
            Enable := FALSE,
            Enable_Positive := FALSE,
            Enable_Negative := FALSE
        );

        nTestStep := nTestStep + 1;
END_CASE

IF nTestStep = 11 THEN
    TEST_FINISHED();
ELSIF fbTestTimer.Q THEN
    AssertTrue(
        Condition := FALSE,
        Message := CONCAT('Timed out at step: ', TO_STRING(nTestStep))
    );

    TEST_FINISHED();
END_IF
END_METHOD

END_FUNCTION_BLOCK

// ---- Tests/PRG_TEST.TcPOU
PROGRAM PRG_TEST
VAR
    fb_AtPositionState_Test: FB_AtPositionState_Test;
    fb_AxisParameterSetExposed_Test: FB_AxisParameterSetExposed_Test;
    fb_MiscStatesErrorFFO_Test: FB_MiscStatesErrorFFO_Test;
    {attribute 'TcNcAxis' := '
        .AxisReference := Axis_MotionAxisNC_Test
    '}
    fbMotionAxisNC_Test : FB_MotionAxisNC_Test;
    {attribute 'TcNcAxis' := '
        .AxisReference := Axis_MotionAxisNCContinuous_Test
    '}
    fbMotionAxisNCContinuous_Test : FB_MotionAxisNCContinuous_Test;
    fb_MotionBPTM_Test: FB_MotionBPTM_Test;
    fb_MotionClearAsserts_Test: FB_MotionClearAsserts_Test;
    fb_MotionReadPMPSDBND_Test: FB_MotionReadPMPSDBND_Test;
    fbMotionVirtualFrameTest: FB_MotionVirtualFrame_Test;
    fb_TestHelperSetAndMove_Test: FB_TestHelperSetAndMove_Test;
    fb_PositionStateRead_Test: FB_PositionStateRead_Test;
    fb_PositionStateReadND_Test: FB_PositionStateReadND_Test;
    fb_PositionStateMove_Test: FB_PositionStateMove_Test;
    fb_PositionStateMoveND_Test: FB_PositionStateMoveND_Test;
    fb_PositionStateND_Test: FB_PositionStateND_Test;
    fb_NCErrorFFO_Test: FB_NCErrorFFO_Test;
    fb_StatePMPSEnables_Test: FB_StatePMPSEnables_Test;
    fb_PerMotorFFOND_Test: FB_PerMotorFFOND_Test;
    fb_StatePMPSEnablesND_Test: FB_StatePMPSEnablesND_Test;
    fb_PositionStatePMPSND_Test: FB_PositionStatePMPSND_Test;
    fb_StateSetupHelper_Test: FB_StateSetupHelper_Test;
    fb_TestStateInitTiming: FB_TestStateInitTiming;
    fb_PowerEnableMode_Test: FB_PowerEnableMode_Test;
    fb_MotionBacklashCompensation_Test: FB_MotionBacklashCompensation_Test;
END_VAR


TcUnit.RUN();

END_PROGRAM

// ---- Tests/TestDoubles/FB_MotionAxisNCTestDouble.TcPOU

FUNCTION_BLOCK FB_MotionAxisNCTestDouble IMPLEMENTS I_MotionAxis
VAR
    bPowerEnable : BOOL;
    bPowerEnable_Positive : BOOL;
    bPowerEnable_Negative : BOOL;
    fPowerOverride : LREAL;
    ePowerBufferMode : MC_BufferMode;

    bPowerStatus : BOOL;
    bPowerBusy : BOOL;
    bPowerActive : BOOL;
    bPowerError	: BOOL;
    nPowerErrorID : UDINT;
    sPowerErrorStr : T_MaxString;

    bHaltDone : BOOL;
    bHaltBusy : BOOL;
    bHaltError : BOOL;
    nHaltErrorID : UDINT;

    bMoveAbsoluteDone : BOOL;
    bMoveAbsoluteBusy : BOOL;
    bMoveAbsoluteActive	: BOOL;
    bMoveAbsoluteCommandAborted	: BOOL;
    bMoveAbsoluteError : BOOL;
    nMoveAbsoluteErrorID : UDINT;
    sMoveAbsoluteErrorStr : T_MaxString;

    fMoveAbsolutePosition : LREAL;
    fMoveAbsoluteVelocity : LREAL;
    fMoveAbsoluteAcceleration : LREAL := 0.0;
    fMoveAbsoluteDeceleration : LREAL := 0.0;
    fMoveAbsoluteJerk : LREAL := 0.0;

    fMeasuredPosition : LREAL;

    fSetpointAcceleration : LREAL;
    fSetpointPosition : LREAL;
    fSetpointJerk : LREAL;
    fSetpointVelocity : LREAL;

    nNumberOfTimesMoveAbsoluteExecuteHasRisingEdge : INT;
END_VAR

{warning 'Add method implementation '}
METHOD CalibrateEncValue
END_METHOD

{warning 'Add method implementation '}
METHOD EncSaveRestore
END_METHOD

{warning 'Add property implementation'}
PROPERTY Error : BOOL
GET
END_GET
END_PROPERTY

{warning 'Add property implementation'}
PROPERTY ErrorID : BOOL
GET
END_GET
END_PROPERTY

{warning 'Add method implementation '}
METHOD GearIn
END_METHOD

{warning 'Add method implementation '}
METHOD GearOut
END_METHOD


METHOD GetAxisRef : REFERENCE TO AXIS_REF
END_METHOD

METHOD PUBLIC GetNumberOfTimesMoveAbsoluteExecuteHasRisingEdge : INT

GetNumberOfTimesMoveAbsoluteExecuteHasRisingEdge := THIS^.nNumberOfTimesMoveAbsoluteExecuteHasRisingEdge;
END_METHOD


METHOD PUBLIC GetPowerOverride : LREAL

GetPowerOverride := THIS^.fPowerOverride;
END_METHOD

{warning 'Add method implementation '}
METHOD Halt
VAR_INPUT
    Deceleration	: LREAL := 0.0;
    Jerk	: LREAL := 0.0;
    BufferMode	: MC_BufferMode := .MC_BufferMode.MC_Aborting;
END_VAR
VAR_OUTPUT
    Done	: BOOL;
    Busy	: BOOL;
    Active	: BOOL;
    CommandAborted	: BOOL;
    Error	: BOOL;
    ErrorID	: UDINT;
    ErrorStr	: T_MaxString;
END_VAR
END_METHOD

{warning 'Add property implementation'}
PROPERTY HaltBusy : BOOL
GET
END_GET
END_PROPERTY

{warning 'Add property implementation'}
PROPERTY HaltDone : BOOL
GET
END_GET
END_PROPERTY

{warning 'Add property implementation'}
PROPERTY HaltError : BOOL
GET
END_GET
END_PROPERTY

{warning 'Add property implementation'}
PROPERTY HaltErrorID : UDINT
GET
END_GET
END_PROPERTY

{warning 'Add method implementation '}
METHOD Home
VAR_INPUT
    Position	: LREAL := .DEFAULT_HOME_POSITION;
    HomingMode	: MC_HomingMode := .MC_DefaultHoming;
END_VAR
VAR_OUTPUT
    Done	: BOOL;
    Busy	: BOOL;
    Active	: BOOL;
    CommandAborted	: BOOL;
    Error	: BOOL;
    ErrorID	: UDINT;
    ErrorStr	: T_MaxString;
END_VAR
END_METHOD

{warning 'Add property implementation'}
PROPERTY HomeBusy : BOOL
GET
END_GET
END_PROPERTY

{warning 'Add property implementation'}
PROPERTY HomeDone : BOOL
GET
END_GET
END_PROPERTY

{warning 'Add property implementation'}
PROPERTY MeasuredAcceleration : LREAL
GET
END_GET
END_PROPERTY


PROPERTY MeasuredPosition : LREAL
GET

MeasuredPosition := THIS^.fMeasuredPosition;
END_GET
SET

THIS^.fMeasuredPosition := MeasuredPosition;
END_SET
END_PROPERTY

{warning 'Add property implementation'}
PROPERTY MeasuredVelocity : LREAL
GET
END_GET
END_PROPERTY


METHOD MoveAbsolute
VAR_INPUT
    Position	: LREAL;
    Velocity	: LREAL;
    Acceleration	: LREAL := 0.0;
    Deceleration	: LREAL := 0.0;
    Jerk	: LREAL := 0.0;
    BufferMode	: MC_BufferMode := .MC_BufferMode.MC_Aborting;
END_VAR
VAR_OUTPUT
    Done	: BOOL;
    Busy	: BOOL;
    Active	: BOOL;
    CommandAborted	: BOOL;
    Error	: BOOL;
    ErrorID	: UDINT;
    ErrorStr	: T_MaxString;
END_VAR

nNumberOfTimesMoveAbsoluteExecuteHasRisingEdge := nNumberOfTimesMoveAbsoluteExecuteHasRisingEdge + 1;
END_METHOD

{warning 'Add property implementation'}
PROPERTY MoveAbsoluteBusy : BOOL
GET

MoveAbsoluteBusy := bMoveAbsoluteBusy;
END_GET
END_PROPERTY


PROPERTY MoveAbsoluteDone : BOOL
GET

MoveAbsoluteDone := bMoveAbsoluteDone;
END_GET
END_PROPERTY


PROPERTY MoveAbsoluteError : BOOL
GET

MoveAbsoluteError := bMoveAbsoluteError;
END_GET
END_PROPERTY


PROPERTY MoveAbsoluteErrorID : UDINT
GET

MoveAbsoluteErrorID := nMoveAbsoluteErrorID;
END_GET
END_PROPERTY

{warning 'Add property implementation'}
PROPERTY MoveAbsoluteTargetAcceleration : LREAL
GET
END_GET
END_PROPERTY

{warning 'Add property implementation'}
PROPERTY MoveAbsoluteTargetDeceleration : LREAL
GET
END_GET
END_PROPERTY

{warning 'Add property implementation'}
PROPERTY MoveAbsoluteTargetJerk : LREAL
GET
END_GET
END_PROPERTY

{warning 'Add property implementation'}
PROPERTY MoveAbsoluteTargetPosition : LREAL
GET
END_GET
END_PROPERTY

{warning 'Add property implementation'}
PROPERTY MoveAbsoluteTargetVelocity : LREAL
GET
END_GET
END_PROPERTY

{warning 'Add property implementation'}
PROPERTY MoveBusy : BOOL
GET
END_GET
END_PROPERTY

{warning 'Add property implementation'}
PROPERTY MoveDone : BOOL
GET
END_GET
END_PROPERTY

{warning 'Add property implementation'}
PROPERTY NegativeMotionIsEnabled : BOOL
GET
END_GET
END_PROPERTY

{warning 'Add property implementation'}
PROPERTY PositionSetpoint : LREAL
GET
END_GET
END_PROPERTY

{warning 'Add property implementation'}
PROPERTY PositiveMotionIsEnabled : BOOL
GET
END_GET
END_PROPERTY


METHOD Power
VAR_INPUT
    Enable	: BOOL;
    Enable_Positive	: BOOL;
    Enable_Negative	: BOOL;
    (* in percent from 0 to 100 *)
    Override	: LREAL := 100.0;
    BufferMode	: MC_BufferMode := .MC_BufferMode.MC_Aborting;
END_VAR
VAR_OUTPUT
    Status	: BOOL;
    Busy	: BOOL;
    Active	: BOOL;
    Error	: BOOL;
    ErrorID	: UDINT;
    ErrorStr	: T_MaxString;
END_VAR

bPowerEnable := Enable;
bPowerEnable_Positive := Enable_Positive;
bPowerEnable_Negative := Enable_Negative;
fPowerOverride := Override;
ePowerBufferMode := BufferMode;

Status := bPowerStatus;
Busy := bPowerBusy;
Active := bPowerActive;
Error := bPowerError;
ErrorID := nPowerErrorID;
ErrorStr := sPowerErrorStr;
END_METHOD


PROPERTY PowerError : BOOL
GET

PowerError := bPowerError;
END_GET
END_PROPERTY


PROPERTY PowerErrorID : UDINT
GET

PowerErrorID := nPowerErrorID;
END_GET
END_PROPERTY

{warning 'Add property implementation'}
PROPERTY PowerIsEnabled : BOOL
GET
END_GET
END_PROPERTY

{warning 'Add property implementation'}
PROPERTY PowerOverride : LREAL
GET
END_GET
END_PROPERTY


PROPERTY PowerStatus : BOOL
GET

PowerStatus := bPowerStatus;
END_GET
END_PROPERTY


METHOD Reset
VAR_OUTPUT
    Done	: BOOL;
    Busy	: BOOL;
    Error	: BOOL;
    ErrorID	: UDINT;
    ErrorStr	: T_MaxString;
END_VAR
END_METHOD

{warning 'Add property implementation'}
PROPERTY ResetBusy : BOOL
GET
END_GET
END_PROPERTY

{warning 'Add property implementation'}
PROPERTY ResetDone : BOOL
GET
END_GET
END_PROPERTY

{warning 'Add property implementation'}
PROPERTY ResetError : BOOL
GET
END_GET
END_PROPERTY

{warning 'Add property implementation'}
PROPERTY ResetErrorID : UDINT
GET
END_GET
END_PROPERTY


METHOD PUBLIC SetMoveAbsoluteOutput
VAR_INPUT
    Done : BOOL;
    Busy : BOOL;
    Active : BOOL;
    CommandAborted : BOOL;
    Error : BOOL;
    ErrorID : UDINT;
    ErrorStr : T_MaxString;
END_VAR

bMoveAbsoluteDone := Done;
bMoveAbsoluteBusy := Busy;
bMoveAbsoluteActive	:= Active;
bMoveAbsoluteCommandAborted	:= CommandAborted;
bMoveAbsoluteError := Error;
nMoveAbsoluteErrorID := ErrorID;
sMoveAbsoluteErrorStr := ErrorStr;
END_METHOD


PROPERTY SetpointAcceleration : LREAL
GET

SetpointAcceleration := fSetpointAcceleration;
END_GET
SET

fSetpointAcceleration := SetpointAcceleration;
END_SET
END_PROPERTY


PROPERTY SetpointJerk : LREAL
GET

SetpointJerk := fSetpointJerk;
END_GET
SET

fSetpointJerk := SetpointJerk;
END_SET
END_PROPERTY


PROPERTY SetpointPosition : LREAL
GET

SetpointPosition := fSetpointPosition;
END_GET
SET

fSetpointPosition := SetpointPosition;
END_SET
END_PROPERTY


PROPERTY SetpointVelocity : LREAL
GET

SetpointVelocity := fSetpointVelocity;
END_GET
SET

fSetpointVelocity := SetpointVelocity;
END_SET
END_PROPERTY


METHOD SetPowerOutput
VAR_INPUT
    Status	: BOOL;
    Busy	: BOOL;
    Active	: BOOL;
    Error	: BOOL;
    ErrorID	: UDINT;
    ErrorStr	: T_MaxString;
END_VAR

bPowerStatus := Status;
bPowerBusy := Busy;
bPowerActive := Active;
bPowerError := Error;
nPowerErrorID := ErrorID;
sPowerErrorStr := ErrorStr;
END_METHOD


METHOD SetPowerOverride
VAR_INPUT
    (* in percent from 0 to 100 *)
    Override : LREAL;
END_VAR
VAR_OUTPUT
    Status : BOOL;
    Busy : BOOL;
    Active : BOOL;
    Error : BOOL;
    ErrorID : UDINT;
    ErrorStr : T_MaxString;
END_VAR

THIS^.fPowerOverride := Override;
END_METHOD

END_FUNCTION_BLOCK
